cart10_front_temp														:= F_Temperature(_10_TT_01, cart10_front_temp_offset);
cart10_front_temp_error 												:= _10_TT_01_error OR iCount[18] < 30;
cart10_back_temp														:= F_Temperature(_10_TT_03, cart10_back_temp_offset);
cart10_back_temp_error 													:= _10_TT_03_Error OR iCount[19] < 30;
cart10_temp_front_calc(Error:= cart10_front_temp_error, Temp:= cart10_front_temp, Low:= sorbent_low_temp, High:= sorbent_high_temp, Total:= rTempTotal, Counter:= iTempCount);
cart10_temp_back_calc(Error:= cart10_back_temp_error, Temp:= cart10_back_temp, Low:= sorbent_low_temp, High:= sorbent_high_temp, Total:= rTempTotal, Counter:= iTempCount);

cart11_front_temp														:= F_Temperature(_11_TT_01, cart11_front_temp_offset);
cart11_front_temp_error 												:= _11_TT_01_error OR iCount[20] < 30;
cart11_back_temp														:= F_Temperature(_11_TT_03, cart11_back_temp_offset);
cart11_back_temp_error 													:= _11_TT_03_Error OR iCount[21] < 30;
cart11_temp_front_calc(Error:= cart11_front_temp_error, Temp:= cart11_front_temp, Low:= sorbent_low_temp, High:= sorbent_high_temp, Total:= rTempTotal, Counter:= iTempCount);
cart11_temp_back_calc(Error:= cart11_back_temp_error, Temp:= cart11_back_temp, Low:= sorbent_low_temp, High:= sorbent_high_temp, Total:= rTempTotal, Counter:= iTempCount);

cart12_front_temp														:= F_Temperature(_12_TT_01, cart12_front_temp_offset);
cart12_front_temp_error 												:= _12_TT_01_error OR iCount[22] < 30;
cart12_back_temp														:= F_Temperature(_12_TT_03, cart12_back_temp_offset);
cart12_back_temp_error 													:= _12_TT_03_Error OR iCount[23] < 30;
cart12_temp_front_calc(Error:= cart12_front_temp_error, Temp:= cart12_front_temp, Low:= sorbent_low_temp, High:= sorbent_high_temp, Total:= rTempTotal, Counter:= iTempCount);
cart12_temp_back_calc(Error:= cart12_back_temp_error, Temp:= cart12_back_temp, Low:= sorbent_low_temp, High:= sorbent_high_temp, Total:= rTempTotal, Counter:= iTempCount);

sorbent_average_temp													:= SEL(iTempCount > 0, 0, rTempTotal / iTempCount);

FOR i:= 0 TO 23 DO
	iCount[i]															:= iCount[i] + 1;
	IF iCount[i] > 30 THEN
		iCount[i]														:= 30;
	END_IF
END_FOR

iHighTempCount															:= 0;
rMin																	:= P_U01.SP_minimum_reasonable_sorbent_TC_reading;
rMax																	:= P_U01.SP_maximum_reasonable_sorbent_TC_reading;
IF iInletAirSetpoint = 0 THEN
	rTempSP																:= P_M01.SP_vacuum_cooling_target_temperature;
ELSIF iInletAirSetpoint = 1 THEN
	rTempSP																:= P_M01.SP_maximum_inlet_air_temperature_during_adsorption;
ELSE
	rTempSP																:= P_M01.SP_maximum_sorbent_temperature_during_desorption;
END_IF

IF _01_TT_01_Error OR cart01_front_temp < rMin OR cart01_front_temp > rMax THEN
	iCount[0]															:= 0;
ELSIF cart01_front_temp > rTempSP THEN
	iHighTempCount														:= iHighTempCount + 1;
END_IF 
IF _01_TT_03_Error OR cart01_back_temp < rMin OR cart01_back_temp > rMax THEN
	iCount[1]															:= 0;
ELSIF cart01_back_temp > rTempSP THEN
	iHighTempCount														:= iHighTempCount + 1;
END_IF

IF _02_TT_01_Error OR cart02_front_temp < rMin OR cart02_front_temp > rMax THEN
	iCount[2]															:= 0;
ELSIF cart02_front_temp > rTempSP THEN
	iHighTempCount														:= iHighTempCount + 1;
END_IF 
IF _02_TT_03_Error OR cart02_back_temp < rMin OR cart02_back_temp > rMax THEN
	iCount[3]															:= 0;
ELSIF cart02_back_temp > rTempSP THEN
	iHighTempCount														:= iHighTempCount + 1;
END_IF

IF _03_TT_01_Error OR cart03_front_temp < rMin OR cart03_front_temp > rMax THEN
	iCount[4]															:= 0;
ELSIF cart03_front_temp > rTempSP THEN
	iHighTempCount														:= iHighTempCount + 1;
END_IF 
IF _03_TT_03_Error OR cart03_back_temp < rMin OR cart03_back_temp > rMax THEN
	iCount[5]															:= 0;
ELSIF cart03_back_temp > rTempSP THEN
	iHighTempCount														:= iHighTempCount + 1;
END_IF

IF _04_TT_01_Error OR cart04_front_temp < rMin OR cart04_front_temp > rMax THEN
	iCount[6]															:= 0;
ELSIF cart04_front_temp > rTempSP THEN
	iHighTempCount														:= iHighTempCount + 1;
END_IF 
IF _04_TT_03_Error OR cart04_back_temp < rMin OR cart04_back_temp > rMax THEN
	iCount[7]															:= 0;
ELSIF cart04_back_temp > rTempSP THEN
	iHighTempCount														:= iHighTempCount + 1;
END_IF

IF _05_TT_01_Error OR cart05_front_temp < rMin OR cart05_front_temp > rMax THEN
	iCount[8]															:= 0;
ELSIF cart05_front_temp > rTempSP THEN
	iHighTempCount														:= iHighTempCount + 1;
END_IF 
IF _05_TT_03_Error OR cart05_back_temp < rMin OR cart05_back_temp > rMax THEN
	iCount[9]															:= 0;
ELSIF cart05_back_temp > rTempSP THEN
	iHighTempCount														:= iHighTempCount + 1;
END_IF

IF _06_TT_01_Error OR cart06_front_temp < rMin OR cart06_front_temp > rMax THEN
	iCount[10]															:= 0;
ELSIF cart06_front_temp > rTempSP THEN
	iHighTempCount														:= iHighTempCount + 1;
END_IF 
IF _06_TT_03_Error OR cart06_back_temp < rMin OR cart06_back_temp > rMax THEN
	iCount[11]															:= 0;
ELSIF cart06_back_temp > rTempSP THEN
	iHighTempCount														:= iHighTempCount + 1;
END_IF

IF _07_TT_01_Error OR cart07_front_temp < rMin OR cart07_front_temp > rMax THEN
	iCount[12]															:= 0;
ELSIF cart07_front_temp > rTempSP THEN
	iHighTempCount														:= iHighTempCount + 1;
END_IF 
IF _07_TT_03_Error OR cart07_back_temp < rMin OR cart07_back_temp > rMax THEN
	iCount[13]															:= 0;
ELSIF cart07_back_temp > rTempSP THEN
	iHighTempCount														:= iHighTempCount + 1;
END_IF

IF _08_TT_01_Error OR cart08_front_temp < rMin OR cart08_front_temp > rMax THEN
	iCount[14]															:= 0;
ELSIF cart08_front_temp > rTempSP THEN
	iHighTempCount														:= iHighTempCount + 1;
END_IF 
IF _08_TT_03_Error OR cart08_back_temp < rMin OR cart08_back_temp > rMax THEN
	iCount[15]															:= 0;
ELSIF cart08_back_temp > rTempSP THEN
	iHighTempCount														:= iHighTempCount + 1;
END_IF

IF _09_TT_01_Error OR cart09_front_temp < rMin OR cart09_front_temp > rMax THEN
	iCount[16]															:= 0;
ELSIF cart09_front_temp > rTempSP THEN
	iHighTempCount														:= iHighTempCount + 1;
END_IF 
IF _09_TT_03_Error OR cart09_back_temp < rMin OR cart09_back_temp > rMax THEN
	iCount[17]															:= 0;
ELSIF cart09_back_temp > rTempSP THEN
	iHighTempCount														:= iHighTempCount + 1;
END_IF

IF _10_TT_01_Error OR cart10_front_temp < rMin OR cart10_front_temp > rMax THEN
	iCount[18]															:= 0;
ELSIF cart10_front_temp > rTempSP THEN
	iHighTempCount														:= iHighTempCount + 1;
END_IF 
IF _10_TT_03_Error OR cart10_back_temp < rMin OR cart10_back_temp > rMax THEN
	iCount[19]															:= 0;
ELSIF cart10_back_temp > rTempSP THEN
	iHighTempCount														:= iHighTempCount + 1;
END_IF

IF _11_TT_01_Error OR cart11_front_temp < rMin OR cart11_front_temp > rMax THEN
	iCount[20]															:= 0;
ELSIF cart11_front_temp > rTempSP THEN
	iHighTempCount														:= iHighTempCount + 1;
END_IF 
IF _11_TT_03_Error OR cart11_back_temp < rMin OR cart11_back_temp > rMax THEN
	iCount[21]															:= 0;
ELSIF cart11_back_temp > rTempSP THEN
	iHighTempCount														:= iHighTempCount + 1;
END_IF

IF _12_TT_01_Error OR cart12_front_temp < rMin OR cart12_front_temp > rMax THEN
	iCount[22]															:= 0;
ELSIF cart12_front_temp > rTempSP THEN
	iHighTempCount														:= iHighTempCount + 1;
END_IF 
IF _12_TT_03_Error OR cart12_back_temp < rMin OR cart12_back_temp > rMax THEN
	iCount[23]															:= 0;
ELSIF cart12_back_temp > rTempSP THEN
	iHighTempCount														:= iHighTempCount + 1;
END_IF

IF iInletAirSetpoint = 0 THEN
	vacuum_cooling_high_temp_count										:= iHighTempCount;
ELSIF iInletAirSetpoint = 1 THEN
	adsorption_high_temp_count											:= iHighTempCount;
ELSE
	desorption_high_temp_count											:= iHighTempCount;
END_IF
iInletAirSetpoint														:= SEL(iInletAirSetpoint = 2, iInletAirSetpoint + 1, 0);;
END_ACTION

END_FUNCTION_BLOCK

// ---- POUs/Function_Blocks/FB_VFD.TcPOU
FUNCTION_BLOCK FB_VFD
VAR_INPUT
	Enable_Vfd															: BOOL;
	Fault_Reset															: BOOL;
	Rpm																	: REAL;
	Minimum_Speed														: REAL		:= 0;
	Maximum_Speed														: REAL		:= 1800;
	StatusWord															: WORD;
END_VAR
VAR_OUTPUT
	ControlWord															: WORD;
	TargetRpm															: WORD;
	Ready																: BOOL;
	Error																: BOOL;
END_VAR
VAR
	rtrigClear															: R_TRIG;
	rtrigReady															: R_TRIG;
	rtrigRun															: R_TRIG;
	tonReady															: TON;
	tonRun																: TON;
	rRpm																: REAL;
	bEnabled															: BOOL;
	
	VFD_OFF																: WORD										:= 0;
	VFD_CLEAR															: WORD										:= 6;
	VFD_READY															: WORD										:= 7;
	VFD_RUN																: WORD										:= 15;
	VFD_FAULTED															: WORD										:= 8;
	VFD_RESET															: WORD										:= 128;
END_VAR

//// FB_VFD
//// Rev 1.0 - April 11, 2024

// Need to add parse status word

rRpm := Rpm;

bEnabled																:= Enable_Vfd;
IF rRpm = 0 THEN
	bEnabled															:= FALSE;											// Turn output off if rpm is 0
ELSIF rRpm > Maximum_Speed THEN
	rRpm																:= Maximum_Speed;
ELSIF rRpm < Minimum_Speed THEN
	rRpm																:= Minimum_Speed;
END_IF

rtrigClear(CLK:= bEnabled);
IF rtrigClear.Q THEN
	ControlWord															:= VFD_CLEAR;
END_IF

rtrigReady(CLK:= tonReady.Q);
IF rtrigReady.Q THEN
	ControlWord															:= VFD_READY;
END_IF
tonReady(IN:= ControlWord = VFD_CLEAR, PT:= T#100MS);

rtrigRun(CLK:= tonRun.Q);
IF rtrigRun.Q THEN
	ControlWord															:= VFD_RUN;
END_IF
tonRun(IN:= ControlWord = VFD_READY, PT:= T#100MS);

IF NOT bEnabled AND NOT Fault_Reset THEN
	ControlWord															:= VFD_OFF;
	rtrigReady(CLK:= FALSE);
END_IF

IF Error AND Fault_Reset THEN
	ControlWord															:= VFD_RESET;
END_IF

Ready																	:= ControlWord = VFD_READY OR ControlWord = VFD_RUN OR Enable_Vfd;
TargetRpm																:= SEL(Ready, 0, REAL_TO_WORD(rRpm));

Error																	:= (StatusWord AND VFD_FAULTED) > 0;

END_FUNCTION_BLOCK

// ---- POUs/Function_Blocks/FB_Door_Closed.TcPOU
FUNCTION_BLOCK FB_Door_Closed
VAR_INPUT
	valve																: BOOL;
	limit_switch														: BOOL;
END_VAR
VAR_OUTPUT
	door_closed															: BOOL;
END_VAR
VAR
	ton1																: TON;
	rtrig1																: R_TRIG;
END_VAR

// FB_Door_Closed
// Rev 1.0 - November 2, 2024

ton1(IN:= valve AND limit_switch, PT:= _DOOR_LATCH_CLOSE_TIME);
rtrig1(CLK:= ton1.Q);
IF rtrig1.Q THEN
	door_closed															:= TRUE;
ELSIF NOT valve THEN
	door_closed															:= FALSE;
END_IF

END_FUNCTION_BLOCK

// ---- POUs/Function_Blocks/FB_Temperature.TcPOU
FUNCTION_BLOCK FB_Temperature
VAR_INPUT
	Error																: BOOL;
	Temp																: REAL;
	Low																	: REFERENCE TO REAL;
	High																: REFERENCE TO REAL;
	Total																: REFERENCE TO REAL;
	Counter																: REFERENCE TO INT;
END_VAR
VAR
END_VAR

// Theseus - FB_Temperature
// Rev 1.0 - April 25, 2024

IF NOT Error THEN
	Low																	:= F_LowestReal(Temp, Low);
	High																:= F_HighestReal(Temp, High, 0, 0);
	Total																:= Total + Temp;
	Counter																:= Counter + 1;
END_IF

END_FUNCTION_BLOCK

// ---- POUs/Functions/F_HighestReal.TcPOU
FUNCTION F_HighestReal : REAL
VAR_INPUT
	Value1																: REAL;
	Value2																: REAL;
	Value3																: REAL;
	Value4																: REAL;
END_VAR
VAR
	rValue																: REAL;
END_VAR

// F_HighestReal
// Rev 1.0 - April 25, 2024

rValue																		:= SEL(Value1 > Value2, Value2, Value1);
rValue																		:= SEL(rValue > Value3, Value3, rValue);
F_HighestReal																:= SEL(rValue > Value4, Value4, rValue);

END_FUNCTION

// ---- POUs/MAIN.TcPOU
PROGRAM MAIN
VAR
	bHalfSecondPulse													: BOOL;
	tonHalfSecPulse														: TON;
END_VAR

// Theseus - Main
// Rev 1.0 - September 31, 2024

P_M01.plc_version														:= '24_12_03_00';

/// TIMER PULSE
IF tonHalfSecPulse.Q THEN
	bHalfSecondPulse													:= NOT bHalfSecondPulse;
	tonHalfSecPulse(IN:= FALSE);
END_IF
tonHalfSecPulse(IN:= TRUE, PT:= T#500MS);

P_U01();
P_M01();
P_Alarms();

END_PROGRAM

// ---- POUs/P_M01.TcPOU
PROGRAM P_M01
VAR_INPUT
	rs1																	: FB_Reactor_Set();
	stop_rs																: BOOL;
	clear_rs															: BOOL;
	
	{attribute 'OPC.UA.DA' := '1'}  				                
	{attribute 'OPC.UA.DA.Access' := '1'}  				                
	plc_version															: STRING;
	{attribute 'OPC.UA.DA' := '1'}  				                
	{attribute 'OPC.UA.DA.Access' := '1'}  				                
	tb_Alarm_Active														: BOOL;			// An alarm is active
	{attribute 'OPC.UA.DA' := '1'}  				                
	{attribute 'OPC.UA.DA.Access' := '1'}  				                
	ts_Alarm															: STRING;		// Active alarm string
	{attribute 'OPC.UA.DA' := '1'}  				                
	{attribute 'OPC.UA.DA.Access' := '1'}  				                
	ts_User_Message														: STRING;		// Message corresponding to active alarm
	{attribute 'OPC.UA.DA' := '1'}  				                
	{attribute 'OPC.UA.DA.Access' := '1'}  				                
	ti_Alarm_Severity													: INT;			// Alarm level (not implemented)	
	{attribute 'OPC.UA.DA' := '1'}  
	processAlarms														: ARRAY[0.._ALARM_COUNT] OF STRING;
	{attribute 'OPC.UA.DA' := '1'}  
	processAlarmsMessage												: ARRAY[0.._ALARM_COUNT] OF STRING;
	{attribute 'OPC.UA.DA' := '1'}  				                
	tb_Acknowledge_Alarm												: BOOL;			// Clears current alarm
	{attribute 'OPC.UA.DA' := '1'}  				                
	tb_Clear_Alarm_All													: BOOL;			// Clears current alarm
END_VAR
VAR
	sCycleModeRS01														: STRING	:= '';
	iRS01CyclesToRun													: INT;
	iLength																: INT;
	iRS01Count															: INT;
	rtrigStart															: R_TRIG;
	
	bRSProcess															: BOOL;
	bRSManual															: BOOL;
	bRS01																: BOOL;
	bRS01Selected														: BOOL;
	bStarted															: BOOL;
	bReactorSetSelected													: BOOL;
	
	rtrigRS01StartNextRS												: R_TRIG;
	rtrigRS01Restart													: R_TRIG;
	rtrigRS01Done														: R_TRIG;
	rtrigRS01Offline													: R_TRIG;
	
	rtrigCPDrainLSHOn													: R_TRIG;
	tonCPDrainErrorOn													: TON;
	tonCPDrainErrorOff													: TON;
	bCPDrainError														: BOOL;
	
	rMinPressureSP														: REAL; 
	rMaxPressureSP														: REAL;
	
	{attribute 'OPC.UA.DA' := '1'}  				                
	ts_Cycle_Mode														: STRING;		// Starts process based on each character in integer format
	{attribute 'OPC.UA.DA' := '1'}  				                
	tb_HMI_Active														: BOOL;			// An HMI program is running and communicating
	{attribute 'OPC.UA.DA' := '1'}  				                
	tb_Cancel_Cycle														: BOOL;			// Complete current cycle then stop
	{attribute 'OPC.UA.DA' := '1'}  				                
	tb_Stop_Process														: BOOL;			// Stop current process immediately
	{attribute 'OPC.UA.DA' := '1'}  				                
	tb_Reset_Process													: BOOL;
	
					
	{attribute 'OPC.UA.DA' := '1'}  				                
	{attribute 'OPC.UA.DA.Access' := '1'}  				                
	tb_Auto_Mode_On														: BOOL;			// Machine is currently in auto mode

END_VAR

VAR PERSISTENT

	/// SET POINTS

	{attribute 'OPC.UA.DA' := '1'}
	SP_evacuation_ideal_pressure										: REAL;
	{attribute 'OPC.UA.DA' := '1'}
	SP_evacuation_duration												: REAL;
	{attribute 'OPC.UA.DA' := '1'}
	SP_vacuum_settle_time												: REAL;
	{attribute 'OPC.UA.DA' := '1'}
	SP_vacuum_leak_test_duration										: REAL;
	{attribute 'OPC.UA.DA' := '1'}
	SP_unacceptable_vacuum_pressure_change								: REAL;
	{attribute 'OPC.UA.DA' := '1'}
	SP_pos_pres_ideal_pressure											: REAL;		
	{attribute 'OPC.UA.DA' := '1'}
	SP_pos_pres_settle_time												: REAL;		
	{attribute 'OPC.UA.DA' := '1'}
	SP_pos_pres_leak_test_duration										: REAL;		
	{attribute 'OPC.UA.DA' := '1'}
	SP_unacceptable_pos_pres_change										: REAL;		

	
	{attribute 'OPC.UA.DA' := '1'}
	SP_adsorption_sorbent_hightemp_startco2analyzer						: REAL;		
	{attribute 'OPC.UA.DA' := '1'}
	SP_adsorption_outletco2_highlimit									: REAL;		
	{attribute 'OPC.UA.DA' := '1'}
	SP_repres_preslimit_clampsretract									: REAL;		
	{attribute 'OPC.UA.DA' := '1'}
	SP_clampsretract_timedelay											: REAL;		
	{attribute 'OPC.UA.DA' := '1'}
	SP_repres_pres_highlimit											: REAL;		
	{attribute 'OPC.UA.DA' := '1'}
	SP_doorsopenclose_timedelay											: REAL;		
	{attribute 'OPC.UA.DA' := '1'}
	SP_adsorption_duration												: REAL;
	{attribute 'OPC.UA.DA' := '1'}
	SP_adsorption_valve_max_retries										: INT;		
	{attribute 'OPC.UA.DA' := '1'}
	SP_adsorption_valve_rotational_velocity								: REAL;		
	{attribute 'OPC.UA.DA' := '1'}
	SP_ambient_pressure													: REAL;
	{attribute 'OPC.UA.DA' := '1'}
	SP_cycle_start_offset_duration										: REAL;
	{attribute 'OPC.UA.DA' := '1'}
	SP_dead_time_in_cycle_duration										: REAL;
	{attribute 'OPC.UA.DA' := '1'}
	SP_desired_cycle_count												: INT;
	{attribute 'OPC.UA.DA' := '1'}
	SP_evacuation_unacceptable_pressure									: REAL;
	{attribute 'OPC.UA.DA' := '1'}
	SP_include_reactor_set_1_in_process									: BOOL;					
	{attribute 'OPC.UA.DA' := '1'}
	SP_include_reactor_set_2_in_process									: BOOL;
	{attribute 'OPC.UA.DA' := '1'}
	SP_include_reactor_set_3_in_process									: BOOL;	
	{attribute 'OPC.UA.DA' := '1'}
	SP_initial_maximum_steam_valve_percent_open							: REAL;
	{attribute 'OPC.UA.DA' := '1'}
	SP_initial_steam_purge_reactor_pressure								: REAL;
	{attribute 'OPC.UA.DA' := '1'}
	SP_leak_test_duration												: REAL;
	{attribute 'OPC.UA.DA' := '1'}
	SP_maximum_desorption_starting_pressure								: REAL;							
	{attribute 'OPC.UA.DA' := '1'}
	SP_maximum_inlet_air_temperature_during_adsorption					: REAL;						
	{attribute 'OPC.UA.DA' := '1'}
	SP_maximum_reactor_leakage_pressure									: REAL;												// PS 11/27/24
	{attribute 'OPC.UA.DA' := '1'}
	SP_maximum_reactor_pressure_to_introduce_steam						: REAL;												// PS 08_12_24
	{attribute 'OPC.UA.DA' := '1'}
	SP_maximum_safe_ambient_temperature									: REAL;												// PS 08_12_24
	{attribute 'OPC.UA.DA' := '1'}
	SP_maximum_safe_co2_adsorption_sensor_temperature					: REAL;												// PS 08_16_24
	{attribute 'OPC.UA.DA' := '1'}
	SP_maximum_safe_reactor_steam_pressure								: REAL;
	{attribute 'OPC.UA.DA' := '1'}
	SP_maximum_safe_sorbent_temperature									: REAL;												// PS 08_15_24
	{attribute 'OPC.UA.DA' := '1'}
	SP_maximum_sorbent_temperature_during_desorption					: REAL;			
	{attribute 'OPC.UA.DA' := '1'}
	SP_maximum_sorbent_temperature_to_use_dead_air_line					: REAL;												// PS 08_12_24			
	{attribute 'OPC.UA.DA' := '1'}
	SP_maximum_target_sorbent_temperature_during_purge					: REAL;												// PS 04_25_24			
	{attribute 'OPC.UA.DA' := '1'}
	SP_maximum_target_sorbent_temperature_to_repressurize				: REAL;												// PS 08_15_24		
	{attribute 'OPC.UA.DA' := '1'}
	SP_maximum_target_steam_pressure									: REAL;			
	{attribute 'OPC.UA.DA' := '1'}
	SP_minimum_desired_inlet_co2_concentration_during_adsorption		: REAL;						
	{attribute 'OPC.UA.DA' := '1'}
	SP_minimum_inlet_air_temperature_during_adsorption					: REAL;						
	{attribute 'OPC.UA.DA' := '1'}
	SP_module_steam_line_high_pressure									: REAL;
	{attribute 'OPC.UA.DA' := '1'}
	SP_module_steam_line_high_temperature								: REAL;
	{attribute 'OPC.UA.DA' := '1'}
	SP_module_steam_line_low_pressure									: REAL;
	{attribute 'OPC.UA.DA' := '1'}
	SP_module_steam_line_low_temperature								: REAL;
	{attribute 'OPC.UA.DA' := '1'}
	SP_percent_from_steam_purge_target_pressure							: REAL;
	{attribute 'OPC.UA.DA' := '1'}
	SP_percent_of_ambient_pressure										: REAL;
	{attribute 'OPC.UA.DA' := '1'}
	SP_reactor_set_1_vfd_percent										: INT;
	{attribute 'OPC.UA.DA' := '1'}
	SP_reactor_set_2_vfd_percent										: INT;
	{attribute 'OPC.UA.DA' := '1'}
	SP_reactor_set_3_vfd_percent										: INT;
	{attribute 'OPC.UA.DA' := '1'}
	SP_repressurization_duration										: REAL;
	{attribute 'OPC.UA.DA' := '1'}
	SP_start_steam_purge_reactor_pressure								: REAL;
	{attribute 'OPC.UA.DA' := '1'}
	SP_steam_pressure_control_valve_initial_opening_duration			: REAL;					
	{attribute 'OPC.UA.DA' := '1'}
	SP_steam_pressurization_and_purge_duration							: REAL;						
	{attribute 'OPC.UA.DA' := '1'}
	SP_steam_purge_pressure												: REAL;
	{attribute 'OPC.UA.DA' := '1'}
	SP_steam_purge_pressure_decrease									: REAL;												// PS 04_25_24
	{attribute 'OPC.UA.DA' := '1'}
	SP_target_desorption_starting_pressure								: REAL;
	{attribute 'OPC.UA.DA' := '1'}
	SP_target_duration_from_adsorption_start_until_sorbent_cool			: REAL;							
	{attribute 'OPC.UA.DA' := '1'}
	SP_target_pressure_change											: REAL;
	{attribute 'OPC.UA.DA' := '1'}
	SP_unacceptable_duration_from_adsorption_start_until_sorbent_cool	: REAL;					
	{attribute 'OPC.UA.DA' := '1'}
	SP_undesirable_duration_from_adsorption_start_until_sorbent_cool	: REAL;
	{attribute 'OPC.UA.DA' := '1'}
	SP_vacuum_assisted_purge											: BOOL;
	{attribute 'OPC.UA.DA' := '1'}
	SP_vacuum_cooling_duration											: REAL;
	{attribute 'OPC.UA.DA' := '1'}
	SP_vacuum_cooling_target_pressure									: REAL;
	{attribute 'OPC.UA.DA' := '1'}
	SP_vacuum_cooling_target_temperature								: REAL;
	{attribute 'OPC.UA.DA' := '1'}
	SP_vacuum_cooling_unacceptable_pressure								: REAL;
	{attribute 'OPC.UA.DA' := '1'}
	SP_vacuum_cooling_unacceptable_temperature							: REAL;
	{attribute 'OPC.UA.DA' := '1'}
	SP_extend_wallace_clamp_duration									: REAL;
			
END_VAR

// Theseus - P_M01
// Rev 1.0 - November 27, 2024

A_Drain_Condensate_Product_Cooling_Lines();

rs1(	stop_rs_automode												:= stop_rs,
        clear_reactor_set_pause											:= clear_rs);
		
rMinPressureSP															:= SP_ambient_pressure - (SP_percent_of_ambient_pressure / 100 * SP_ambient_pressure); 
rMaxPressureSP															:= SP_ambient_pressure + (SP_percent_of_ambient_pressure / 100 * SP_ambient_pressure);

A_AutoMode();

ACTION A_AutoMode:
// Theseus - P_M01.A_AutoMode
// Rev 1.0 - October 4, 2024

IF tb_Stop_Process OR rs1.utility_error THEN 																	// Stop all processes from HMI or if utility error occurs
	P_U01.shutdown_process												:= TRUE;
//	rs1.stop_rs_automode												:= TRUE;
	stop_rs																:= TRUE;
	bRSProcess															:= FALSE;
	tb_Stop_Process														:= FALSE;
END_IF

IF tb_Cancel_Cycle OR rs1.cancel_all_reactor_sets THEN
	iRS01CyclesToRun													:= SEL(rs1.tb_Process_Running, iRS01Count, iRS01Count + 1);
	bRS01																:= SEL(iRS01Count >= iRS01CyclesToRun, bRS01, FALSE);
	tb_Cancel_Cycle														:= FALSE;
END_IF

A_AutoMode_RS01();

bReactorSetSelected														:= SP_include_reactor_set_1_in_process;
IF ts_Cycle_Mode <> '' AND (P_U01.sUtilityError <> '' OR SP_desired_cycle_count = 0 OR NOT bReactorSetSelected) THEN		// Don't allow cycle if moodule or utility error occured, cycle count is zero or no reactor sets are selected
	IF P_U01.sUtilityError  <> '' THEN
		P_Alarms.M_Add_Alarm(_U01, P_U01.sUtilityError, gsProcessCannotRun);
	ELSIF SP_desired_cycle_count = 0 THEN
		P_Alarms.M_Add_Alarm(_U01, gsDesiredCycleCountError, gsProcessCannotRun);
	ELSE
		P_Alarms.M_Add_Alarm(_U01, gsNoReactorSetsSelected, gsProcessCannotRun);
	END_IF
	ts_Cycle_Mode														:= '';
END_IF

iLength																	:= LEN(ts_Cycle_Mode);							// Start process in this order '6745' (Evac, Desorp, Repres, Adsorp)
rtrigStart(CLK:= iLength > 0);
IF rtrigStart.Q THEN
	gsCycleMode															:= ts_Cycle_Mode;
	ts_Cycle_Mode														:= '';
	iRS01CyclesToRun													:= SP_desired_cycle_count;
	bRS01																:= SP_include_reactor_set_1_in_process;			// Get active reactors
	IF iLength = 1 THEN																										// Single process selected
		tb_Auto_Mode_On													:= FALSE;
		bRSManual														:= STRING_TO_INT(gsCycleMode) >= eDoorCycle AND STRING_TO_INT(gsCycleMode) <= eDesorption;
	ELSE
		bRS01Selected													:= bRS01;
		rs1.ti_Cycle_Count												:= 0;												// Completed cycles
		iRS01Count														:= 0;												// Attempted cycles
		tb_Auto_Mode_On													:= TRUE;
		bRSProcess														:= TRUE;
	END_IF
END_IF

IF bRSManual THEN
	sCycleModeRS01														:= SEL(bRS01, sCycleModeRS01, gsCycleMode);
	bRSManual															:= FALSE;
ELSIF bRSProcess THEN
	IF NOT bStarted THEN
		sCycleModeRS01													:= gsCycleMode;
		bStarted														:= TRUE;
	END_IF
	IF NOT bRS01 THEN																										// Stop process if reactor is not selected
//		rs1.stop_rs_automode											:= TRUE;
		stop_rs															:= TRUE;
		bRSProcess														:= FALSE;
	END_IF
	
	rtrigRS01Done(CLK:= rs1.Done);
	IF rtrigRS01Done.Q THEN
		sCycleModeRS01													:= '';												// Turn off cycle
		bStarted														:= FALSE;
		iRS01Count														:= iRS01Count + 1;									// This counter increments regardless of reactor status if long as reactor was selected
		IF iRS01Count >= iRS01CyclesToRun THEN
			bRS01														:= FALSE;
			gsCycleMode													:= '';
		END_IF
		IF rs1.tb_Process_Complete THEN 																				// Increment counter once a valid cycle has run
			rs1.ti_Cycle_Count											:= rs1.ti_Cycle_Count + 1;
			rs1.ti_Total_Cycle_Count									:= 1;			///@@@
		END_IF
	END_IF
	
ELSE
//	P_U01.write_persistent_data											:= TRUE;
	sCycleModeRS01														:= '';
	bRS01																:= FALSE;
	bStarted															:= FALSE;
	tb_Auto_Mode_On														:= FALSE;
	
END_IF

rs1.cycle_mode 															:= sCycleModeRS01;

IF NOT rs1.Process_Running THEN 
	rs1.cycle_stage														:= gsCycleStage;
//	gsCycleMode															:= '';
END_IF

// rs1.cycle_stage															:= SEL(bRS01 AND gsCycleStage <> '', gsM01RS01CycleStage, gsCycleStage);
END_ACTION

ACTION A_AutoMode_RS01:
// Theseus - P_M01.A_AutoMode_RS01
// Rev 1.0 - October 4, 2024

rtrigRS01Restart(CLK:= SP_include_reactor_set_1_in_process);
IF rtrigRS01Restart.Q THEN
	IF tb_Auto_Mode_On AND NOT bRS01Selected THEN 
		SP_include_reactor_set_1_in_process								:= FALSE;
	ELSE
		bRS01															:= TRUE;
		rs1.clear_rs_pause												:= TRUE;
	END_IF
END_IF

//IF rs1.stop_rs_automode THEN
IF stop_rs THEN
	SP_include_reactor_set_1_in_process									:= FALSE;
	bRS01Selected														:= FALSE;
END_IF

rtrigRS01Offline(CLK:= NOT SP_include_reactor_set_1_in_process);
IF rtrigRS01Offline.Q THEN
	bRS01																:= FALSE;
END_IF

IF rs1.cancel_reactor_set THEN
	iRS01CyclesToRun													:= SEL(rs1.tb_Process_Running, iRS01Count, iRS01Count + 1);
END_IF
END_ACTION

ACTION A_Drain_Condensate_Product_Cooling_Lines:
// Theseus - P_M01.A_Drain_Condensate_Product_Cooling_Lines
// Rev 1.0 - June 10, 2024

(*IF gbDrainageOn THEN
	IF (P_U01.purge_product_line_pres < P_U01.SP_drainage_function_cutoff_pressure) OR
		(m01_rs1.purge_valve_closed AND m01_rs1.condensate_valve_closed) THEN
		m.condensate_from_cooling_and_purge_lines_pump					:= FALSE;
	ELSE
		IF m.condensate_from_cooling_and_purge_linesh THEN
			m.condensate_from_cooling_and_purge_lines_pump				:= TRUE;
		END_IF
		IF NOT m.condensate_from_cooling_and_purge_linesl THEN
			m.condensate_from_cooling_and_purge_lines_pump				:= FALSE;
		END_IF
	END_IF
	
	rtrigCPDrainLSHOn(CLK:= tonCPDrainErrorOn.Q);
	IF rtrigCPDrainLSHOn.Q THEN
		P_Alarms.M_Add_Alarm(_M01, gsCondensateProductDrainError, gsProcessStopsAtEOC);
		m.condensate_from_cooling_and_purge_lines_pump					:= FALSE;
		bCPDrainError													:= TRUE;
		m01.tb_Cancel_Cycle												:= TRUE;											// Complete current cycles
	END_IF
	tonCPDrainErrorOn(IN:= m.condensate_from_cooling_and_purge_linesh AND NOT bCPDrainError, PT:= _DRAIN_TIME);
	
	IF tonCPDrainErrorOff.Q THEN
		bCPDrainError													:= FALSE;
	END_IF
	tonCPDrainErrorOff(IN:= NOT m.condensate_from_cooling_and_purge_linesh AND bCPDrainError, PT:= _DRAIN_TIME);
END_IF
*)
END_ACTION

END_PROGRAM

// ---- POUs/FB_Reactor_Set.TcPOU
FUNCTION_BLOCK FB_Reactor_Set
VAR_IN_OUT
	//stop_reactor_set													: BOOL;
	stop_rs_automode													: BOOL;
	clear_reactor_set_pause												: BOOL;
END_VAR
VAR_INPUT
	r1																	: FB_Reactor;
	
	rs_name																: STRING;
	cycle_mode															: STRING;
//	stop_rs_automode													: BOOL;
	clear_rs_pause														: BOOL;
	open_doors															: BOOL;
	close_doors															: BOOL;
	close_valves														: BOOL;
	retract_clamps														: BOOL;
	extend_clamps														: BOOL;
	
	{attribute 'OPC.UA.DA' := '1'}  				                
	fan_setpoint														: REAL;
	{attribute 'OPC.UA.DA' := '1'}  				                
	{attribute 'OPC.UA.DA.Access' := '1'}  				                
	ti_Cycle_Count														: INT; 
	{attribute 'OPC.UA.DA' := '1'}  				                
	{attribute 'OPC.UA.DA.Access' := '1'}  				                
	ti_Total_Cycle_Count												: DINT; 
	{attribute 'OPC.UA.DA' := '1'}  				                
	{attribute 'OPC.UA.DA.Access' := '1'}  				                
	cycle_stage															: STRING;
    /// <summary>RS_XV08</summary>
	{attribute 'OPC.UA.DA' := '1'}  				                
	steam_bypass_valve													: BOOL;
	/// <summary>XV02</summary>
	{attribute 'OPC.UA.DA' := '1'}  	//mm 11/7 to command valve
	repres_valves														: BOOL;
END_VAR
VAR_OUTPUT
	
	inlet_doors_open													: BOOL;
	inlet_doors_closed													: BOOL;
	outlet_doors_open													: BOOL;
	outlet_doors_closed													: BOOL;

	inlet_clamps_extended												: BOOL;
	inlet_clamps_retracted												: BOOL;
	outlet_clamps_extended												: BOOL;
	outlet_clamps_retracted												: BOOL;
	
	rs_valves_clear														: BOOL;
	adsorption_high_temp_count											: INT;
	desorption_high_temp_count											: INT;
	vacuum_cooling_high_temp_count										: INT;
	sorbent_high_temp													: REAL;
	sorbent_average_temp												: REAL;
	
    /// <summary>Reactor XV02</summary>
	repres_valves_clear													: BOOL;
    /// <summary>RS_XV04</summary>
	dead_air_valve_clear												: BOOL;
    /// <summary>RS_XV05</summary>
	product_iso_valve_clear												: BOOL;
    /// <summary>RS_XV06</summary>
	condensate_valve_clear												: BOOL;
    /// <summary>RS_XV07</summary>
	steam_iso_valve_clear												: BOOL;
    /// <summary>RS_XV08</summary>
	steam_bypass_valve_clear											: BOOL;
	
	/// <summary>RS_LS01</summary>
	{attribute 'OPC.UA.DA' := '1'}  				                
	{attribute 'OPC.UA.DA.Access' := '1'}  				                
	reactor_drain_vessel_lsl									AT %I*	: BOOL;
    /// <summary>RS_LS02</summary>
	{attribute 'OPC.UA.DA' := '1'}  				                
	{attribute 'OPC.UA.DA.Access' := '1'}  				                
	reactor_drain_vessel_lsh									AT %I*	: BOOL;

    /// <summary>RS_FT02</summary>
	{attribute 'OPC.UA.DA' := '1'}  				                
	{attribute 'OPC.UA.DA.Access' := '1'}  				                
	reactor_condensate_flow												: REAL;

	Remaining_Time														: REAL;
	Current_Step														: INT;
	Machine_State														: INT;
	Status																: INT;
	Process_Running														: BOOL;
	Pause_Reactor_Set													: BOOL;
	Reactor_Set_Stopped													: BOOL;
	DoorCycle_Running													: BOOL;
	PositivePressure_Running											: BOOL;
	Repressurization_Running											: BOOL;
	Adsorption_Running													: BOOL;
	Evacuation_Running													: BOOL;
	Desorption_Running													: BOOL;
	Bypass_Running														: BOOL;
	Utility_Error														: BOOL;
	Cancel_Reactor_Set													: BOOL;
	Cancel_All_Reactor_Sets												: BOOL;
	Process_Complete													: BOOL;
	Done																: BOOL;
	
END_VAR
VAR
	eState																: E_MachineState;
	i																	: INT;
	iStatePointer														: INT;
	iLength																: INT;
	iStateMode															: ARRAY[0..9] OF INT;
	stop_reactor_set													: BOOL;
	
	sUtilityError														: STRING;
	sReactorError														: STRING;
	sCancelError														: STRING;
	sRetryError															: STRING;
	sError																: STRING;
	sMessage															: STRING;
	sLeakageAcceptable													: STRING;
	sLeakageUnacceptable												: STRING;

	rAveragePressure													: REAL;
	iCount																: INT;
	iVacuumStatus														: INT;
	iError																: INT;
	
	rTime																: REAL;
	rTime1																: REAL;
	rTime2																: REAL;
	rTime3																: REAL;
	rSP1																: REAL;
	rSP2																: REAL;
	rSP3																: REAL;
	rR1SavedPressure													: REAL;
	rR1Leakage															: REAL;
	rIncrementalMove													: REAL;
	rPosition															: REAL;
	rAverageReactorPres													: REAL;
	rReactorLeakTestStartingPressure									: REAL;
	
	tTime																: TIME;
	
	iStep																: INT;
	i2Step																: INT;
	i3Step																: INT;
	i4Step																: INT;
	i5Step																: INT;
	i6Step																: INT;
	i7Step																: INT;
	i8Step																: INT;
	iStartStep															: INT;
	iStatus																: INT;
	iErrorProcess														: INT;
	iR1Leakage															: INT;
	iCycleCount															: INT;
	iMaxSorbentTempErrorCount											: INT;

	bMultiProcess														: BOOL;
	bEndProcess															: BOOL;
	bSPAdjust															: BOOL;
	bPaused																: BOOL;
	bClearingCycle														: BOOL;
	bDoorCycleDone								        				: BOOL;
	bPositivePressureDone						        				: BOOL;
	bRepressurizationDone												: BOOL;
	bAdsorptionDone														: BOOL;
	bEvacuationDone														: BOOL;
	bDesorptionDone									        			: BOOL;
	bBypassDone									        				: BOOL;
	bPass1																: BOOL;
	bPass2																: BOOL;
	bPass3																: BOOL;
	bPass4																: BOOL;
	bPass5																: BOOL;
	bPass6																: BOOL;
	bPass7																: BOOL;
	bPass8																: BOOL;
	bPass9																: BOOL;
	bPass10																: BOOL;
	
	
	bCondenserKnockoutOn												: BOOL;
	bStop																: BOOL;
	bTimer1																: BOOL;
	bTimer2																: BOOL;
	bTimer3																: BOOL;
	bRunning															: BOOL;
	bDrainError															: BOOL;
	bPumpOn																: BOOL;
	bPumpTimeOut														: BOOL;									
	bDrainResetToLSL													: BOOL;
	bProcessStarted														: BOOL;
	bDesorptionErrorCheck												: BOOL;
	bSafeShutdownOn														: BOOL;
	bInletClampsRetracted												: BOOL;
	bInletClampsExtended												: BOOL;
	bOutletClampsRetracted												: BOOL;
	bOutletClampsExtended												: BOOL;
	bVacuumHolding														: BOOL;
	bCondition21														: BOOL;
	bCondition22														: BOOL;
	bCondition11														: BOOL;
	bCondition12														: BOOL;
	
	rtrigStart															: R_TRIG;
	rtrigPaused															: R_TRIG;
	rtrigIdle															: R_TRIG;
	rtrigDoorCycle														: R_TRIG;
	rtrigPositivePressure												: R_TRIG;
	rtrigRepressurization												: R_TRIG;
	rtrigAdsorption														: R_TRIG;
	rtrigEvacuation														: R_TRIG;
	rtrigDesorption														: R_TRIG;
	rtrigBypass															: R_TRIG;
	rtrigSingleProcessAuto												: R_TRIG;
	rtrigDrainLSHOn														: R_TRIG;
	
	tonTimer1															: TON;
	tonTimer2															: TON;
	tonTimer3															: TON;
	tonPause															: TON;
	tonDrain															: TON;
	rtrigCondensateValveOff_DrainOff									: R_TRIG;
	tonProcess															: TON;
	
	tRestartTime														: TIME;

	bSteamHeaderValve													: BOOL;
	bCondition1															: BOOL;
	bCondition2															: BOOL;
	bCondition3															: BOOL;
	
	reactor_drain_adsorption_on											: BOOL;
	tmrDrainAdsorp														: TON;
	waterscale_desorp													: REAL;
	water_scale_change_oor												: BOOL;
	fb_adsorp_reactor_wastewater											: FB_ChangeOfValue;
	
	
	{attribute 'OPC.UA.DA' := '1'}  				                
	{attribute 'OPC.UA.DA.Access' := '1'}  				                
	ti_Machine_State													: INT;
	{attribute 'OPC.UA.DA' := '1'}  				                
	{attribute 'OPC.UA.DA.Access' := '1'}  				                
	ti_Current_Step														: INT;
	{attribute 'OPC.UA.DA' := '1'}  				                
	{attribute 'OPC.UA.DA.Access' := '1'}  				                
	tb_Process_Running													: BOOL;
	{attribute 'OPC.UA.DA' := '1'}  				                
	{attribute 'OPC.UA.DA.Access' := '1'}  				                
	tb_Repressurization_Running											: BOOL;
	{attribute 'OPC.UA.DA' := '1'}  				                
	{attribute 'OPC.UA.DA.Access' := '1'}  				                
	tb_Adsorption_Running												: BOOL;
	{attribute 'OPC.UA.DA' := '1'}  				                
	{attribute 'OPC.UA.DA.Access' := '1'}  				                
	tb_Evacuation_Running												: BOOL;
	{attribute 'OPC.UA.DA' := '1'}  				                
	{attribute 'OPC.UA.DA.Access' := '1'}  				                
	tb_Desorption_Running												: BOOL;
	{attribute 'OPC.UA.DA' := '1'}  				                
	{attribute 'OPC.UA.DA.Access' := '1'}  				                
	tb_Bypass_Running													: BOOL;
	{attribute 'OPC.UA.DA' := '1'}  				                
	{attribute 'OPC.UA.DA.Access' := '1'}  				                
	tb_Process_Complete													: BOOL;
	{attribute 'OPC.UA.DA' := '1'}  				                
	{attribute 'OPC.UA.DA.Access' := '1'}  				                
	tr_Remaining_Time													: REAL;
	{attribute 'OPC.UA.DA' := '1'}  				                
	{attribute 'OPC.UA.DA.Access' := '1'}  				                
	ti_Status															: INT;
	{attribute 'OPC.UA.DA' := '1'}  				                
	{attribute 'OPC.UA.DA.Access' := '1'}  				                
	ts_Status_Text														: STRING;		

	

	{attribute 'OPC.UA.DA' := '1'}  				                
	{attribute 'OPC.UA.DA.Access' := '1'}  				                
	interlock_inlet_door_clamps_or										: BOOL;

	{attribute 'OPC.UA.DA' := '1'}  				                
	{attribute 'OPC.UA.DA.Access' := '1'}  				                
	interlock_outlet_door_clamps_or										: BOOL;

	{attribute 'OPC.UA.DA' := '1'}  				                
	interlock_inlet_door_or												: BOOL;
	{attribute 'OPC.UA.DA' := '1'} 		      
	{attribute 'OPC.UA.DA.Access' := '1'}  				                
	interlock_inlet_door_or_status										: BOOL;
	{attribute 'OPC.UA.DA' := '1'}  				                
	{attribute 'OPC.UA.DA.Access' := '1'}  				                
	interlock_outlet_door_or											: BOOL;
	{attribute 'OPC.UA.DA' := '1'}  				                
	{attribute 'OPC.UA.DA.Access' := '1'}  				                
	interlock_outlet_door_or_status										: BOOL;
	
	{attribute 'OPC.UA.DA' := '1'}  				                
	interlock_inlet_door_clamp_or										: BOOL;
	{attribute 'OPC.UA.DA' := '1'}  				                
	{attribute 'OPC.UA.DA.Access' := '1'}  				                
	interlock_inlet_door_clamp_or_status								: BOOL;
	{attribute 'OPC.UA.DA' := '1'}  						                
	interlock_outlet_door_clamp_or										: BOOL;
	{attribute 'OPC.UA.DA' := '1'}  				                
	{attribute 'OPC.UA.DA.Access' := '1'}  				                
	interlock_outlet_door_clamp_or_status								: BOOL;
	
    /// <summary>PWR-01</summary>
	{attribute 'OPC.UA.DA' := '1'}  				                
	power_control														: BOOL;
    /// <summary>PWR-01</summary>
	{attribute 'OPC.UA.DA' := '1'}  				                
	{attribute 'OPC.UA.DA.Access' := '1'}  				                
	power_control_status												: BOOL;
    /// <summary>power_cmd</summary>
	PWR_01														AT %Q*	: BOOL;
	circuit_breaker_no_feedback									AT %I*	: BOOL;
	circuit_breaker_nc_feedback									AT %I*	: BOOL;
	

    /// <summary>RS_TT01</summary>
	{attribute 'OPC.UA.DA' := '1'}  				                
	{attribute 'OPC.UA.DA.Access' := '1'}  				                
	product_line_temp													: REAL;
    /// <summary>RS_TT01</summary>
	{attribute 'OPC.UA.DA' := '1'}  				                
	{attribute 'OPC.UA.DA.Access' := '1'}
	product_line_temp_error												: BOOL;
    /// <summary>RS_TT01</summary>
	{attribute 'OPC.UA.DA' := '1'}  				                
	_ProductLineTempErrorOff											: BOOL		:= TRUE;
    /// <summary>rs product line temp</summary>
	TT_01														AT %I*	: INT;
    /// <summary>rs product line temp</summary>
	TT_01_error													AT %I*	: BOOL;
	
    /// <summary>RS_PT02</summary>
	{attribute 'OPC.UA.DA' := '1'}  				                
	{attribute 'OPC.UA.DA.Access' := '1'}  				                
	product_line_pres													: REAL;
    /// <summary>RS_PT02</summary>
	{attribute 'OPC.UA.DA' := '1'}  				                
	{attribute 'OPC.UA.DA.Access' := '1'}  				                
	product_line_pres_error												: BOOL;
    /// <summary>RS_PT02</summary>
	{attribute 'OPC.UA.DA' := '1'}  				                
	_ProductLinePresErrorOff											: BOOL;
    /// <summary>rs product line temp</summary>
	PT_02														AT %I*	: INT;
    /// <summary>rs product line temp</summary>
	PT_02_error													AT %I*	: BOOL;
	
    /// <summary>RS_FT02</summary>
	{attribute 'OPC.UA.DA' := '1'}  				                
	{attribute 'OPC.UA.DA.Access' := '1'}  				                
	reactor_condensate_flow_error										: BOOL;
    /// <summary>RS_FT02</summary>
	{attribute 'OPC.UA.DA' := '1'}  				                
	_ReactorCondensateFlowErrorOff										: BOOL;
    /// <summary>rs reactor condensate flow</summary>
	FT_02														AT %I*	: INT;
    /// <summary>rs reactor condensate flow</summary>
	FT_02_error													AT %I*	: BOOL;

    /// <summary>RS_XV04</summary>
	{attribute 'OPC.UA.DA' := '1'}  				                
	dead_air_valve														: BOOL;
    /// <summary>RS_XV04</summary>
	{attribute 'OPC.UA.DA' := '1'}  				                
	{attribute 'OPC.UA.DA.Access' := '1'}  				                
	dead_air_valve_open_cmd_status										: BOOL;
    /// <summary>RS_XV04</summary>
	{attribute 'OPC.UA.DA' := '1'}  				                
	{attribute 'OPC.UA.DA.Access' := '1'}  				                
	dead_air_valve_open											AT %I*	: BOOL;
    /// <summary>RS_XV04</summary>
	{attribute 'OPC.UA.DA' := '1'}  				                
	{attribute 'OPC.UA.DA.Access' := '1'}  				                
	dead_air_valve_closed										AT %I*	: BOOL;
    /// <summary>dead air valve</summary>
	XV_04														AT %Q*	: BOOL;
	
    /// <summary>RS_XV05</summary>
	{attribute 'OPC.UA.DA' := '1'}  				                
	product_iso_valve													: BOOL;
    /// <summary>RS_XV05</summary>
	{attribute 'OPC.UA.DA' := '1'}  				                
	{attribute 'OPC.UA.DA.Access' := '1'}  				                
	product_iso_valve_open_cmd_status									: BOOL;
    /// <summary>RS_XV05</summary>
	{attribute 'OPC.UA.DA' := '1'}  				                
	{attribute 'OPC.UA.DA.Access' := '1'}  				                
	product_iso_valve_open										AT %I*	: BOOL;
    /// <summary>RS_XV05</summary>
	{attribute 'OPC.UA.DA' := '1'}  				                
	{attribute 'OPC.UA.DA.Access' := '1'}  				               
	product_iso_valve_closed									AT %I*	: BOOL;
    /// <summary>rs product iso valve</summary>
	XV_05														AT %Q*	: BOOL;
	
     /// <summary>RS_XV06</summary>
	{attribute 'OPC.UA.DA' := '1'}  				                
	condensate_valve													: BOOL;
    /// <summary>RS_XV06</summary>
	{attribute 'OPC.UA.DA' := '1'}  				                
	{attribute 'OPC.UA.DA.Access' := '1'}  				                
	condensate_valve_open_cmd_status									: BOOL;
    /// <summary>RS_XV06</summary>
	{attribute 'OPC.UA.DA' := '1'}  				                
	{attribute 'OPC.UA.DA.Access' := '1'}  				                
	condensate_valve_open										AT %I*	: BOOL;
    /// <summary>RS_XV06</summary>
	{attribute 'OPC.UA.DA' := '1'}  				                
	{attribute 'OPC.UA.DA.Access' := '1'}  				                
	condensate_valve_closed										AT %I*	: BOOL;
    /// <summary>cooling valve</summary>
	XV_06														AT %Q*	: BOOL;
	
    /// <summary>RS_XV07</summary>
	{attribute 'OPC.UA.DA' := '1'}  				                
	steam_iso_valve														: BOOL;
    /// <summary>RS_XV07</summary>
	{attribute 'OPC.UA.DA' := '1'}  				                
	{attribute 'OPC.UA.DA.Access' := '1'}  				                
	steam_iso_valve_open_cmd_status										: BOOL;
    /// <summary>RS_XV07</summary>
	{attribute 'OPC.UA.DA' := '1'}  				                
	{attribute 'OPC.UA.DA.Access' := '1'}  				                
	steam_iso_valve_closed										AT %I*	: BOOL;
    /// <summary>RS_XV07</summary>
	{attribute 'OPC.UA.DA' := '1'}  				                
	{attribute 'OPC.UA.DA.Access' := '1'}  				                
	steam_iso_valve_open										AT %I*	: BOOL;
    /// <summary>steam isolation valve</summary>
	XV_07														AT %Q*	: BOOL;

    /// <summary>RS_XV08</summary>
	{attribute 'OPC.UA.DA' := '1'}  				                
	{attribute 'OPC.UA.DA.Access' := '1'}  				                
	steam_bypass_valve_open_cmd_status									: BOOL;
    /// <summary>RS_XV08</summary>
	{attribute 'OPC.UA.DA' := '1'}  				                
	{attribute 'OPC.UA.DA.Access' := '1'}  				                
	steam_bypass_valve_open										AT %I*	: BOOL;
    /// <summary>RS_XV08</summary>
	{attribute 'OPC.UA.DA' := '1'}  				                
	{attribute 'OPC.UA.DA.Access' := '1'}  				                
	steam_bypass_valve_closed									AT %I*	: BOOL;
    /// <summary>steam bypass valve</summary>
	XV_08														AT %Q*	: BOOL;

	{attribute 'OPC.UA.DA' := '1'}  				                
	{attribute 'OPC.UA.DA.Access' := '1'}  				                
	reactor_test_leakage_pressure										: REAL;

END_VAR
VAR PERSISTENT
	
	{attribute 'OPC.UA.DA' := '1'}
	SP_include_inlet_doors_in_process									: BOOL;					
	{attribute 'OPC.UA.DA' := '1'}
	SP_include_outlet_doors_in_process									: BOOL;					

    /// <summary>TT01</summary>
	{attribute 'OPC.UA.DA' := '1'}  				                
	product_line_temp_offset											: REAL;

    /// <summary>PT02</summary>
	{attribute 'OPC.UA.DA' := '1'}  				                
	product_line_pres_low												: REAL;
    /// <summary>PT02</summary>
	{attribute 'OPC.UA.DA' := '1'}  				                
	product_line_pres_high												: REAL;
    /// <summary>PT02</summary>
	{attribute 'OPC.UA.DA' := '1'}  				                
	product_line_pres_min												: REAL;
    /// <summary>PT02</summary>
	{attribute 'OPC.UA.DA' := '1'}  				                
	product_line_pres_offset											: REAL;
	
    /// <summary>RS FT02</summary>
	{attribute 'OPC.UA.DA' := '1'}  				                
	reactor_condensate_flow_low											: REAL;
    /// <summary>RS FT02</summary>
	{attribute 'OPC.UA.DA' := '1'}  				                
	reactor_condensate_flow_high										: REAL;
    /// <summary>RS FT02</summary>
	{attribute 'OPC.UA.DA' := '1'}  				                
	reactor_condensate_flow_min											: REAL;
    /// <summary>RS FT02</summary>
	{attribute 'OPC.UA.DA' := '1'}  				                
	reactor_condensate_flow_offset										: REAL;
	
END_VAR

// Theseus - FB_Reactor_Set
// Rev 1.0 - December 2, 2024

r1(unit := 1);

A_Reactor_Set_IO();

IF eState <> eIdle THEN 
	A_Clear_Variables();
END_IF

iLength																	:= LEN(cycle_mode);
rtrigStart(CLK:= iLength > 0);
IF rtrigStart.Q THEN
	IF cycle_mode = '0' THEN
		bClearingCycle													:= TRUE;											// This acts as if the cycle ran so the reactor set cycle counter will stay in sync with the other reactor sets		
	ELSE
		bProcessStarted													:= TRUE;
		IF Pause_Reactor_Set THEN
			bPaused														:= TRUE;
		ELSE
			iStartStep													:= 1;
			Process_Running												:= TRUE;
			bMultiProcess												:= iLength > 1;
			giEvacuationCounter											:= 0;
			FOR i := 1 TO iLENGTH DO
				iStateMode[i]											:= STRING_TO_INT(MID(cycle_mode, 1, i));
				IF (iStateMode[i] = 6) THEN
					gbFirstEvacuation									:= TRUE;
					giEvacuationCounter									:= giEvacuationCounter + 1;
				END_IF
			END_FOR
			iStatePointer												:= 1;
			Machine_State												:= iStateMode[1];
		END_IF
	END_IF
END_IF

rtrigIdle(				CLK:= eState <= eIdle);
rtrigPaused(			CLk:= bPaused);
rtrigDoorCycle(			CLK:= Machine_State = eDoorCycle);
rtrigSingleProcessAuto(	CLK:= Machine_State = eSingleProcessAuto);
rtrigRepressurization(	CLK:= Machine_State = eRepressurization);
rtrigAdsorption(		CLK:= Machine_State = eAdsorption);
rtrigEvacuation(		CLK:= Machine_State = eEvacuation);
rtrigPositivePressure(	CLK:= Machine_State = ePositivePressure);
rtrigDesorption(		CLK:= Machine_State = eDesorption);
rtrigBypass(			CLK:= Machine_State = eBypass);

IF rtrigPaused.Q THEN
	bPaused																:= FALSE;
	eState																:= ePause;
ELSIF rtrigDoorCycle.Q THEN
	bDoorCycleDone														:= FALSE;
	i2Step																:= iStartStep;
	eState																:= eDoorCycle;
ELSIF rtrigPositivePressure.Q THEN
	bPositivePressureDone												:= FALSE;
	i3Step																:= iStartStep;
	eState																:= ePositivePressure;
ELSIF rtrigRepressurization.Q THEN
	bRepressurizationDone												:= FALSE;
	i4Step																:= iStartStep;
	eState																:= eRepressurization;
ELSIF rtrigAdsorption.Q THEN
	bAdsorptionDone														:= FALSE;
	i5Step																:= iStartStep;
	eState																:= eAdsorption;
ELSIF rtrigEvacuation.Q THEN
	bEvacuationDone														:= FALSE;
	i6Step																:= iStartStep;
	eState																:= eEvacuation;
ELSIF rtrigDesorption.Q THEN
	bDesorptionDone														:= FALSE;
	i7Step																:= iStartStep;
	eState																:= eDesorption;
ELSIF rtrigBypass.Q THEN
	bBypassDone															:= FALSE;
	i8Step																:= iStartStep;
	eState																:= eBypass;
ELSIF rtrigSingleProcessAuto.Q THEN
	eState																:= eSingleProcessAuto;
ELSIF rtrigIdle.Q THEN
	bProcessStarted														:= FALSE;
	eState																:= eIdle;
END_IF

CASE eState OF
	
	eIdle:
		A_Idle();
		
	eDoorCycle:
		IF bDoorCycleDone THEN
			DoorCycle_Running											:= FALSE;
			IF bMultiProcess THEN
				eState													:= SEL(bStop, eChangeState, ePause);
			ELSE
				Status													:= SEL(bStop, eDoorCycle_Complete, Status);
				eState													:= ePause;
			END_IF
		ELSIF bStop THEN
			Status														:= eStopping_Process;
		ELSE
			Status														:= eDoorCycle_Running;
			DoorCycle_Running											:= TRUE;
		END_IF
		
	ePositivePressure:
		IF bPositivePressureDone THEN
			PositivePressure_Running									:= FALSE;
			IF bMultiProcess THEN
				eState													:= SEL(bStop, eChangeState, ePause);
			ELSE
				Status													:= SEL(bStop, ePositivePressure_Complete, Status);
				eState													:= ePause;
			END_IF
		ELSIF bStop THEN
			Status														:= eStopping_Process;
		ELSE
			Status														:= ePositivePressure_Running;
			PositivePressure_Running									:= TRUE;
		END_IF

	eRepressurization:
		IF bRepressurizationDone THEN
			Repressurization_Running									:= FALSE;
			IF bMultiProcess THEN
				eState													:= SEL(bStop, eChangeState, ePause);
			ELSE
				Status													:= SEL(bStop, eRepressurization_Complete, Status);
				eState													:= ePause;
			END_IF
		ELSIF bStop THEN
			Status														:= eStopping_Process;
		ELSE
			Status														:= eRepressurization_Running;
			Repressurization_Running									:= TRUE;
		END_IF

	eAdsorption:
		IF bAdsorptionDone THEN
			Adsorption_Running											:= FALSE;
			IF bMultiProcess THEN
				eState													:= SEL(bStop, eChangeState, ePause);
			ELSE
				Status													:= SEL(bStop, eAdsorption_Complete, Status);
				eState													:= ePause;
			END_IF
		ELSIF bStop THEN
			Status														:= eStopping_Process;
		ELSE
			Status														:= eAdsorption_Running;
			Adsorption_Running											:= TRUE;
		END_IF

	eEvacuation:
		IF bEvacuationDone THEN
			Evacuation_Running											:= FALSE;
			IF bMultiProcess THEN
				eState													:= SEL(bStop, eChangeState, ePause);
			ELSE
				Status													:= SEL(bStop, eEvacuation_Complete, Status);
				eState													:= ePause;
			END_IF
		ELSIF bStop THEN
			Status														:= eStopping_Process;
		ELSE
			Status														:= eEvacuation_Running;
			Evacuation_Running											:= TRUE;
		END_IF
		
	eDesorption:
		IF bDesorptionDone THEN
			Desorption_Running											:= FALSE;
			IF bMultiProcess THEN
				eState													:= SEL(bStop, eChangeState, ePause);
			ELSE
				Status													:= SEL(bStop, eDesorption_Complete, Status);
				eState													:= ePause;
			END_IF
		ELSIF bStop THEN
			Status														:= eStopping_Process;
		ELSE
			Status														:= eDesorption_Running;
			Desorption_Running											:= TRUE;
		END_IF
		
	eBypass:
		IF bBypassDone THEN
			Bypass_Running												:= FALSE;
			IF bMultiProcess THEN
				eState													:= SEL(bStop, eChangeState, ePause);
			ELSE
				Status													:= SEL(bStop, eBypass_Complete, Status);
				eState													:= ePause;
			END_IF
		ELSIF bStop THEN
			Status														:= eStopping_Process;
		ELSE
			Status														:= eBypass_Running;
			Bypass_Running												:= TRUE;
		END_IF
		
	eSingleProcessAuto:
		eState															:= eChangeState;
		
	eChangeState:
		iStatePointer													:= iStatePointer + 1;
		IF iStatePointer > iLength THEN
			Process_Complete											:= TRUE;
			Done														:= TRUE;
			eState														:= eIdle;
		ELSIF iStateMode[iStatePointer] = 0 THEN
			Status														:= eStopping_Process;
			bStop														:= TRUE;
			bMultiProcess												:= FALSE;
			eState														:= ePause;
		ELSE
			Machine_State												:= iStateMode[iStatePointer];
		END_IF
	
	ePause:
		Machine_State													:= ePause;
		IF tonPause.Q THEN
			Done														:= TRUE;
			eState														:= eIdle;
		END_IF
		
END_CASE

bRunning																:= eState >= eRepressurization AND eState <= ePause;

A2_DoorCycle_1();
A3_PositivePressure_1();
A4_Repressurization_1();
A5_Adsorption_1();
A6_Evacuation_1();
A7_Desorption_1();
A8_Bypass_1();

(*
A4_Repressurization();
A5_Adsorption();
A6_Evacuation();
A7_Desorption();
A8_Bypass();
*)


A_Drain_Reactor_Set();

tonTimer1(IN:= bTimer1, PT:= REAL_TO_TIME(rTime1));
tonTimer2(IN:= bTimer2, PT:= REAL_TO_TIME(rTime2));
tonTimer3(IN:= bTimer3, PT:= REAL_TO_TIME(rTime3));

Remaining_Time															:= 0;
IF Process_Running THEN
	IF bTimer1 THEN
		Remaining_Time													:= rTime1 - TIME_TO_REAL(tonTimer1.ET);
	ELSIF bTimer2 THEN
		Remaining_Time													:= rTime2 - TIME_TO_REAL(tonTimer2.ET);
	ELSIF bTimer3 THEN
		Remaining_Time													:= rTime3 - TIME_TO_REAL(tonTimer3.ET);
	END_IF
END_IF

tonPause(IN:= eState = ePause, PT:= _TIMEOUT_RESET);
tonProcess(IN:= bProcessStarted, PT:= T#10H);

ti_Current_Step := Current_Step;
tr_Remaining_Time := Remaining_Time;
tb_Process_Running := Process_Running;

ACTION A_Check_Process:
// Theseus - FB_Reactor_Set.A_ClearProcess
// Rev 1.0 - June 13, 2024

Current_Step															:= iStep;
bEndProcess																:= FALSE;
IF stop_reactor_set THEN																									// Reactor Set can be stopped both internally and externally
	stop_reactor_set													:= FALSE;											// Clear flag
	bEndProcess															:= TRUE;											// Set flag to end process
ELSE
	IF sUtilityError <> '' THEN
		sError															:= sUtilityError;
		Utility_Error													:= TRUE;
		iStep															:= 98;
	ELSIF sReactorError <> '' THEN
		sError															:= sReactorError;
  		bEndProcess														:= TRUE;
	END_IF
	IF sError <> '' THEN
		P_Alarms.M_Add_Alarm(rs_name, F_Concat3(cycle_stage, ' ', sError), sMessage);
		sError															:= '';
	END_IF
END_IF

IF bEndProcess THEN
	bTimer1								 								:= FALSE;
	bTimer2								 								:= FALSE;
	bStop																:= TRUE;
	iStep																:= SEL(bMultiProcess, 80, 90);
END_IF
END_ACTION

ACTION A_Clear_Variables:
// Theseus - FB_Reactor_Set.A_Clear_Variables
// Rev 1.0 - November 26, 2024

//close_all_valves													:= FALSE;
//co2_sensors_on														:= FALSE;
Utility_Error															:= FALSE;
Cancel_Reactor_Set														:= FALSE;
Cancel_All_Reactor_Sets													:= FALSE;
sUtilityError															:= '';
sReactorError															:= '';
sRetryError																:= '';
IF clear_reactor_set_pause THEN
	clear_reactor_set_pause												:= FALSE;
	Pause_Reactor_Set													:= FALSE;
END_IF
IF NOT P_U01.auto_mode_on THEN
	iMaxSorbentTempErrorCount											:= 0;
	iCycleCount															:= 0;	
END_IF
END_ACTION

ACTION A_Drain_Reactor_Set:
// Theseus - FB_Reactor_Set.A_Drain_Reactor_Set
// Rev 1.0 - October 4, 2024

IF (gbDrainageOn OR P_U01.reactor_drain_or_on) AND NOT P_U01.reactor_drain_or_off THEN
	IF NOT r1.reactor_pres_error AND r1.reactor_pres >= P_U01.SP_minimum_drainage_pressure THEN
//		tonDrain(IN:= NOT bDrainError AND condensate_valve, PT:= REAL_TO_TIME(P_U01.SP_maximum_duration_to_drain_reactor_set * _SECONDS));
		IF tonDrain.Q AND reactor_condensate_flow < P_U01.SP_minimum_condensate_flow THEN
			condensate_valve											:= FALSE;
			IF TRUE THEN ///@@@reactor_drain_vessel_high THEN
				P_U01.steam_flow_control_valve							:= _CLOSED;
				P_Alarms.M_Add_Alarm(rs_name, gsReactorDrainError, gsMessageTBD);
				bDrainError												:= TRUE;
			END_IF
		ELSIF reactor_drain_vessel_lsh THEN ///@@@reactor_drain_vessel_high THEN							mm 11/7 
			condensate_valve											:= TRUE;
		ELSIF NOT reactor_drain_vessel_lsh AND NOT reactor_drain_vessel_lsl THEN ///@@@reactor_drain_vessel_low AND NOT reactor_drain_vessel_high THEN
			condensate_valve											:= FALSE;
//			bDrainError													:= FALSE;
		END_IF
	ELSE
//		IF NOT P_U01.reactor_drain_or_off  THEN 
			condensate_valve												:= FALSE;
//		END_IF
	END_IF
END_IF

rtrigCondensateValveOff_DrainOff(CLK := NOT gbDrainageOn AND NOT P_U01.reactor_drain_or_on AND NOT P_U01.reactor_drain_or_off);
IF 	rtrigCondensateValveOff_DrainOff.Q THEN
	condensate_valve												:= FALSE;
END_IF


gbCondensateValve														:= condensate_valve;

fb_adsorp_reactor_wastewater
	( i_execute := reactor_drain_adsorption_on,
	  i_value := P_U01.water_scale_3,
	  i_time := 30,
	  i_threshold := 1);
	  
IF reactor_drain_adsorption_on THEN
	IF NOT fb_adsorp_reactor_wastewater.o_below_threshold THEN
		condensate_valve											:= TRUE;
	ELSIF fb_adsorp_reactor_wastewater.o_below_threshold OR fb_adsorp_reactor_wastewater.o_timeout THEN
		condensate_valve											:= FALSE;
		reactor_drain_adsorption_on := FALSE;
	END_IF
END_IF
END_ACTION

ACTION A_Idle:
// Theseus - FB_Reactor_Set.A_Idle
// Rev 1.0 - June 24, 2024

Machine_State															:= eIdle;
cycle_stage																:= 'idle.idle';
sError																	:= '';
i4Step																	:= 0;
i5Step																	:= 0;
i6Step																	:= 0;
i7Step																	:= 0;
Current_Step															:= 0;
Remaining_Time															:= 0;
Current_Step															:= 0;
Status																	:= 0;
bMultiProcess															:= FALSE;
bTimer1																	:= FALSE;
bTimer2																	:= FALSE;
bStop																	:= FALSE;
Process_Running															:= FALSE;
Process_Complete														:= FALSE;
IF bClearingCycle THEN
	Done																:= TRUE;
	bClearingCycle														:= FALSE;
ELSE
	Done																:= FALSE;
END_IF
END_ACTION

ACTION A_Reactor_Set_IO:
// Theseus - A_Reactor_Set_IO
// Rev 1.0 - November 26, 2024

r1.fan_vfd_setpoint														:= fan_setpoint;

repres_valves_clear														:= r1.repres_valve_clear;

rAverageReactorPres														:= r1.reactor_pres;

//rso_power_control_out													:= rsi_power_control_fdbk_no AND NOT rsi_power_control_fdbk_nc AND NOT rso_PWR_01 ;
//rso_PWR_01																:= rsi_power_control_in;

interlock_inlet_door_or_status											:= interlock_inlet_door_or;
interlock_outlet_door_or_status											:= interlock_outlet_door_or;
interlock_inlet_door_clamp_or_status									:= interlock_inlet_door_clamp_or;
interlock_outlet_door_clamp_or_status									:= interlock_outlet_door_clamp_or;

inlet_doors_open														:= r1.inlet_doors_open;
inlet_doors_closed														:= r1.inlet_doors_closed;
outlet_doors_open														:= r1.outlet_doors_open;
outlet_doors_closed			 											:= r1.outlet_doors_closed;
 
gbGasketsActivated														:= SEL(NOT inlet_doors_closed OR NOT outlet_doors_closed, gbGasketsActivated, FALSE);					// PS 08_20_24

inlet_clamps_extended													:= r1.inlet_door_clamps_extended;
inlet_clamps_retracted													:= r1.inlet_door_clamps_retracted;
outlet_clamps_extended													:= r1.outlet_door_clamps_extended;
outlet_clamps_retracted													:= r1.outlet_door_clamps_retracted;

IF close_valves THEN
	dead_air_valve														:= FALSE;
	product_iso_valve													:= FALSE;
	condensate_valve													:= FALSE;
	steam_iso_valve														:= FALSE;
	steam_bypass_valve													:= FALSE;
	close_valves														:= FALSE;
END_IF

// Interlock 12
P_U01.door_open_with_steam_flow_interlock								:= NOT P_U01.steam_flow_control_valve_closed AND NOT steam_iso_valve_closed;
bCondition21															:= NOT P_U01.interlock_door_open_with_steam_flow_or AND P_U01.door_open_with_steam_flow_interlock;

// Interlock 14
P_U01.door_open_with_reactor_vacuum_interlock							:= rAverageReactorPres < 0.95;
bCondition22															:= NOT P_U01.interlock_door_open_with_reactor_vacuum_or AND P_U01.door_open_with_reactor_vacuum_interlock;

IF open_doors THEN
	r1.open_inlet_door													:= (inlet_clamps_retracted OR interlock_inlet_door_clamp_or)  AND NOT bCondition21 AND NOT bCondition22; // AND SP_include_inlet_doors_in_process;
	r1.open_outlet_door													:= (outlet_clamps_retracted OR interlock_outlet_door_clamp_or)  AND NOT bCondition21 AND NOT bCondition22; // AND SP_include_outlet_doors_in_process;
	open_doors															:= FALSE;
END_IF
IF close_doors THEN
	r1.close_inlet_door													:= (inlet_clamps_retracted OR interlock_inlet_door_clamp_or) ; //AND SP_include_inlet_doors_in_process;
	r1.close_outlet_door												:= (outlet_clamps_retracted OR interlock_outlet_door_clamp_or); // AND SP_include_outlet_doors_in_process;
	close_doors															:= FALSE;
END_IF

IF extend_clamps THEN
	r1.extend_inlet_door_clamps											:= (inlet_doors_closed OR interlock_inlet_door_or) AND SP_include_inlet_doors_in_process;
	r1.extend_outlet_door_clamps										:= (outlet_doors_closed OR interlock_outlet_door_or) AND SP_include_outlet_doors_in_process;
	extend_clamps														:= FALSE;
END_IF
IF retract_clamps THEN
	r1.retract_inlet_door_clamps										:= SP_include_inlet_doors_in_process;
	r1.retract_outlet_door_clamps										:= SP_include_outlet_doors_in_process;
	retract_clamps														:= FALSE;
END_IF

// CO2 adsorption sensor function
P_U01.co2_adsorption_interlock											:= r1.fan_vfd_setpoint > 10 AND r1.sorbent_high_temp < P_M01.SP_maximum_safe_co2_adsorption_sensor_temperature;
IF NOT P_U01.interlock_co2_adsorption_or THEN
	r1.inlet_co2_sol													:= P_U01.co2_adsorption_interlock;
	r1.outlet_co2_sol													:= P_U01.co2_adsorption_interlock;
	r1.outlet_co2_pump													:= TRUE;
	r1.inlet_co2_pump													:= TRUE;
ELSE
	r1.outlet_co2_pump													:= FALSE;
	r1.inlet_co2_pump													:= FALSE;
END_IF


r1.repres_valve															:= repres_valves AND gbRepresValves;

// Interlock 3
P_U01.hot_reactor_condenser_interlock									:= r1.temp_average > P_M01.SP_maximum_sorbent_temperature_to_use_dead_air_line;
IF NOT P_U01.interlock_hot_reactor_condenser_or and P_U01.hot_reactor_condenser_interlock THEN
	dead_air_valve														:= FALSE;
END_IF

XV_04																	:= dead_air_valve;
dead_air_valve_open_cmd_status											:= XV_04;
dead_air_valve_clear													:= F_ValveClear(dead_air_valve, dead_air_valve_open, dead_air_valve_closed);

XV_05																	:= product_iso_valve;
product_iso_valve_open_cmd_status										:= XV_05;
product_iso_valve_clear													:= F_ValveClear(product_iso_valve, product_iso_valve_open, product_iso_valve_closed);

XV_06																	:= condensate_valve;
condensate_valve_open_cmd_status										:= XV_06;
condensate_valve_clear													:= F_ValveClear(condensate_valve, condensate_valve_open, condensate_valve_closed);

// Interlock 4
P_U01.no_steam_unevacuated_reactor_interlock							:= r1.temp_high < P_M01.SP_maximum_safe_ambient_temperature AND NOT P_U01.steam_flow_control_valve_closed AND r1.reactor_pres < P_M01.SP_maximum_reactor_pressure_to_introduce_steam;
bCondition1																:= P_U01.interlock_no_steam_unevacuated_reactor_or OR P_U01.no_steam_unevacuated_reactor_interlock;

// Interlock 10
P_U01.reactor_over_safe_pressure_limit_interlock						:= r1.reactor_pres <= P_M01.SP_maximum_safe_reactor_steam_pressure;
bCondition2																:= P_U01.interlock_reactor_over_safe_pressure_limit_or OR P_U01.reactor_over_safe_pressure_limit_interlock;
r1.over_pressure_test_control											:= SEL(NOT bCondition2, r1.over_pressure_test_control, FALSE);

// Interlock 11
P_U01.reactor_over_safe_temperature_limit_interlock						:= r1.temp_high <= P_M01.SP_maximum_safe_sorbent_temperature;
bCondition3																:= P_U01.interlock_reactor_over_safe_temperature_limit_or OR P_U01.reactor_over_safe_temperature_limit_interlock;

IF NOT bCondition1 OR NOT bCondition2 OR NOT bCondition3 THEN
	steam_iso_valve														:= FALSE;
END_IF

XV_07																	:= steam_iso_valve;
steam_iso_valve_open_cmd_status											:= XV_07;
steam_iso_valve_clear													:= F_ValveClear(steam_iso_valve, steam_iso_valve_open, steam_iso_valve_closed);

XV_08																	:= steam_bypass_valve;
steam_bypass_valve_open_cmd_status										:= XV_08;
steam_bypass_valve_clear												:= F_ValveClear(steam_bypass_valve, steam_bypass_valve_open, steam_bypass_valve_closed);

rs_valves_clear															:= dead_air_valve_clear AND product_iso_valve_clear AND steam_iso_valve_clear AND steam_bypass_valve_clear AND condensate_valve_clear;

product_line_temp														:= F_Temperature(TT_01, product_line_temp_offset);
product_line_temp_error													:= TT_01_error AND NOT _ProductLineTempErrorOff;

product_line_pres														:= F_AnalogIn(PT_02, product_line_pres_low, product_line_pres_high, product_line_pres_min, product_line_pres_offset);
product_line_pres_error													:= PT_02_error AND NOT _ProductLinePresErrorOff;

reactor_condensate_flow													:= F_AnalogIn(FT_02, reactor_condensate_flow_low, reactor_condensate_flow_high, reactor_condensate_flow_min, reactor_condensate_flow_offset);
reactor_condensate_flow_error											:= FT_02_error AND NOT _ReactorCondensateFlowErrorOff;


gbCondenserKODrainageOn													:= product_line_pres >= P_U01.SP_minimum_drainage_pressure;

adsorption_high_temp_count												:= r1.adsorption_high_temp_count;
desorption_high_temp_count												:= r1.desorption_high_temp_count;
vacuum_cooling_high_temp_count											:= r1.vacuum_cooling_high_temp_count;
sorbent_high_temp														:= r1.sorbent_high_temp;
sorbent_average_temp													:= r1.sorbent_average_temp;

stop_reactor_set														:= stop_rs_automode;
stop_rs_automode														:= FALSE;
clear_reactor_set_pause													:= clear_rs_pause;
clear_rs_pause															:= FALSE;

//reactor_over_max_pressure												:= NOT r1.reactor_pres_error AND r1.reactor_pres > P_M01.SP_maximum_safe_reactor_steam_pressure;

rAveragePressure														:= 0;
iCount																	:= 0;
iVacuumStatus															:= 0;
iError																	:= 4;
IF NOT r1.reactor_pres_error THEN
	rAveragePressure													:= rAveragePressure + r1.reactor_pres;
	iVacuumStatus														:= F_LowMidHigh(r1.reactor_pres, P_M01.SP_target_desorption_starting_pressure, P_M01.SP_maximum_desorption_starting_pressure, iVacuumStatus);
	iCount																:= iCount + 1;
	iError																:= iError - 1;
END_IF
END_ACTION

ACTION A_Reset:
// Theseus - FB_Reactor_Set.A_Reset
// Rev 1.0 - November 25, 2024

r1.over_pressure_test_control											:= FALSE;
repres_valves															:= FALSE;
//co2_sensors_on														:= FALSE;
dead_air_valve															:= FALSE;
product_iso_valve														:= FALSE;
condensate_valve														:= FALSE;
steam_iso_valve															:= FALSE;
steam_bypass_valve														:= FALSE;
fan_setpoint															:= 0;
END_ACTION

ACTION A2_DoorCycle_1:
// Theseus - FB_Reactor_Set.A2_DoorCycle_1
// Rev 1.0 - June 26, 2024

CASE i2Step OF	

	0:	;
		
	1:
		cycle_stage														:= 'doorcycle.initialize';
		sMessage														:= gsSystemCannotRun;
		rTime1															:= 5 * _SECONDS;
		i2Step															:= i2Step + 1;
		
	2:
		bTimer1															:= TRUE;
		IF tonTimer1.Q THEN
			bTimer1														:= FALSE;
			i2Step														:= 99;
		END_IF
		
	99:
		bDoorCycleDone													:= TRUE;											// 9
		Current_Step													:= 0;
		i2Step															:= 0;
	
	
END_CASE

IF i2Step > 0 AND i2Step < 80 THEN
	iStep																:= i2Step;
	Current_Step														:= iStep;
	A_Check_Process();
	i2Step																:= iStep;
END_IF
END_ACTION

ACTION A2_DoorCycle_OLD:
// Theseus - FB_Reactor_Set.A2_DoorCycle
// Rev 1.0 - October 9, 2024

CASE i2Step OF	

	0:	;
		
	1:
		cycle_stage														:= 'doorcycle.initialize';
		sMessage														:= gsSystemCannotRun;
		IF NOT SP_include_inlet_doors_in_process AND NOT SP_include_outlet_doors_in_process THEN
			sReactorError												:= gsDoorsNotSelectedError;
		ELSIF r1.reactor_pres_error THEN
			sReactorError												:= gsReactorPresSensorError;
		ELSE
			A_Reset();																										// 1
			rTime1														:= 5 * _SECONDS;
			i2Step														:= i2Step + 1;
		END_IF
		
	2:
		bTimer1															:= TRUE;
		IF r1.reactor_pres > 0.98 AND r1.reactor_pres < 1.02 THEN															// 2
			bTimer1														:= FALSE;
			i2Step														:= i2Step + 1;
		ELSIF tonTimer1.Q THEN
			sReactorError												:= gsReactorNotAtAmbientPressure;
		END_IF
		
	3:
		bTimer1															:= TRUE;
		bPass1															:= bInletClampsRetracted;
		bPass2															:= bOutletClampsRetracted;
		IF bPass1 AND bPass2 THEN																							// 3
			bTimer1														:= FALSE;
			repres_valves												:= TRUE;											// 4
			rTime1														:= _VALVE_TIME;
			i2Step														:= i2Step + 1;
		ELSIF tonTimer1.Q THEN
			sReactorError												:= gsClampsNotRetractedError;
		END_IF
	
	4:
		bTimer1															:= TRUE;
		IF repres_valves_clear THEN
			cycle_stage													:= 'doorcycle.open';
			bTimer1														:= FALSE;
			open_doors													:= TRUE;											// 5
			rTime1														:= _DOOR_ACTUATION_TIMEOUT;
			i2Step														:= i2Step + 1;
		ELSIF tonTimer1.Q THEN
			sReactorError												:= gsRepressurizationValveError;
		END_IF
		
	5:
		bTimer1															:= TRUE;
		IF inlet_doors_open AND outlet_doors_open THEN
			bTimer1														:= FALSE;
			rTime1														:= 5 * _SECONDS;
			i2Step														:= i2Step + 1;
		ELSIF tonTimer1.Q THEN
			sReactorError												:= gsInletDoorNotOpenError;
			sReactorError												:= SEL(inlet_doors_open, gsOutletDoorNotOpenError, sReactorError);
		END_IF
		
	6:
		bTimer1															:= TRUE;
		IF tonTimer1.Q THEN																									// 6
			cycle_stage													:= 'doorcycle.close';
			bTimer1														:= FALSE;
			close_doors													:= TRUE;											// 7
			rTime1														:= _DOOR_ACTUATION_TIMEOUT;
			i2Step														:= i2Step + 1;
		END_IF
		
	7:
		bTimer1															:= TRUE;
		IF inlet_doors_closed AND outlet_doors_closed THEN
			bTimer1														:= FALSE;
			rTime1														:= 5 * _SECONDS;
			i2Step														:= i2Step + 1;
		ELSIF tonTimer1.Q THEN
			sReactorError												:= gsInletDoorNotClosedError;
			sReactorError												:= SEL(bPass2, gsOutletDoorNotClosedError, sReactorError);
		END_IF

	8:		
		bTimer1															:= TRUE;
		IF tonTimer1.Q THEN																									// 8
			bTimer1														:= FALSE;
			i2Step														:= 99;
		END_IF
	
	80:																														// Manual process closing
		cycle_stage														:= 'doorcycle.stopping';
		rTime1															:= _STOPPING_TIME;
		A_Reset();
		i2Step															:= 98;
		
	90:																														// Automatic process stopping
		cycle_stage														:= 'doorcycle.stopping';
		rTime1															:= _STOPPING_TIME;
		A_Reset();
		i2Step															:= 98;
		
	98:
		bTimer1															:= TRUE;
		IF tonTimer1.Q THEN
			bTimer1														:= FALSE;
			i2Step														:= 99;
		END_IF
		
	99:
		bDoorCycleDone													:= TRUE;											// 9
		Current_Step													:= 0;
		i2Step															:= 0;
	
	
END_CASE

IF i2Step > 0 AND i2Step < 80 THEN
	iStep																:= i2Step;
	Current_Step														:= iStep;
	A_Check_Process();
	i2Step																:= iStep;
END_IF
END_ACTION

ACTION A3_PositivePressure_1:
// Theseus - FB_Reactor_Set.A3_PositivePressure_1
// Rev 1.0 - June 26, 2024

CASE i3Step OF	

	0:	;
		
	1:
		cycle_stage														:= 'positivepressure.initialize';
		sMessage														:= gsSystemCannotRun;
		rTime1															:= _VALVE_TIME;
		i3Step															:= i3Step + 1;

	2:
		bTimer1															:= TRUE;
		IF tonTimer1.Q THEN
			bTimer1														:= FALSE;
			i3Step														:= 99;
		END_IF
	
	99:
		bPositivePressureDone											:= TRUE;
		Current_Step													:= 0;
		i3Step															:= 0;
	
	
END_CASE

IF i3Step > 0 AND i3Step < 80 THEN
	iStep																:= i3Step;
	Current_Step														:= iStep;
	A_Check_Process();
	i3Step																:= iStep;
END_IF
END_ACTION

ACTION A3_PositivePressure_OLD:
// Theseus - FB_Reactor_Set.A3_PositivePressure
// Rev 1.0 - October 3, 2024

CASE i3Step OF	

	0:	;
		
	1:
		cycle_stage														:= 'positivepressure.initialize';
		sMessage														:= gsSystemCannotRun;
		IF r1.reactor_pres_error THEN
			sReactorError												:= gsReactorPresSensorError;
		ELSE
			A_Reset();																										// 1
			i3Step														:= i3Step + 1;
		END_IF

	2:
		IF gbGasketsActivated THEN																							// 2
			rTime1														:= _VALVE_TIME;
			i3Step														:= i3Step + 1;
		ELSE
			sReactorError												:= gsGasketNotActivatedError;
		END_IF
		
	3:
		bTimer1															:= TRUE;
		IF repres_valves_clear AND rs_valves_clear THEN																	// 3
			bTimer1														:= FALSE;
			i3Step														:= i3Step + 1;
		ELSIF tonTimer1.Q THEN
			sReactorError												:= gsRepressurizationValveError;
			sReactorError												:= SEL(steam_iso_valve_clear, gsSteamIsoValveError, sReactorError);
			sReactorError												:= SEL(steam_bypass_valve_clear, gsSteamBypassValveError, sReactorError);
			sReactorError												:= SEL(product_iso_valve_clear, gsProductIsoValveError, sReactorError);
			sReactorError												:= SEL(dead_air_valve_clear, gsDeadAirValveError, sReactorError);
			sReactorError												:= SEL(condensate_valve_clear, gsCondensateValveError, sReactorError);
		END_IF
	
	4:
		IF bInletClampsExtended AND bOutletClampsExtended THEN																// 4
			cycle_stage													:= 'positivepressure.pressurizing';
			//m01_rs1_r1.XV_09											:= TRUE;											// smrg debug
			r1.over_pressure_test_control								:= TRUE;
			//overpressure_test_control								:= TRUE;											// 5
			rTime1														:= 5 * _MINUTES;
			i3Step														:= i3Step + 1;
		ELSE
			sReactorError												:= gsClampsNotExtendedError;
		END_IF
		
	5:
		bTimer1															:= TRUE;
		IF r1.reactor_pres >= P_M01.SP_pos_pres_ideal_pressure THEN
			bTimer1														:= FALSE;
			cycle_stage													:= 'positivepressure.settling';
			r1.over_pressure_test_control								:= FALSE;											// 6
			rTime1														:= P_M01.SP_pos_pres_settle_time * _MINUTES;		// 7
			i3Step														:= i3Step + 1;
		ELSIF tonTimer1.Q THEN
			sReactorError												:= gsPositivePressureError;
		END_IF
	
	6:
		bTimer1															:= TRUE;
		IF tonTimer1.Q THEN
			rR1SavedPressure											:= r1.reactor_pres;									// 8
			cycle_stage													:= 'positivepressure.leak_test';
			rTime1														:= P_M01.SP_pos_pres_leak_test_duration * _MINUTES;	// 9
			i3Step														:= i3Step + 1;
		END_IF
		
	7:
		bTimer1															:= TRUE;
		IF tonTimer1.Q THEN
			bTimer1														:= FALSE;
			rR1Leakage													:= (r1.reactor_pres - rR1SavedPressure) / P_M01.SP_pos_pres_leak_test_duration;	// 10
			IF rR1Leakage > P_M01.SP_unacceptable_pos_pres_change THEN
				sReactorError											:= gsUnacceptableReactorLeakRate;
			ELSE
				i3Step													:= 99;												// 11
			END_IF
		END_IF
		
	80:																														// Manual process closing
		cycle_stage														:= 'positivePressure.stopping';
		rTime1															:= _STOPPING_TIME;
		A_Reset();
		i3Step															:= 98;
		
	90:																														// Automatic process stopping
		cycle_stage														:= 'positivePressure.stopping';
		rTime1															:= _STOPPING_TIME;
		A_Reset();
		i3Step															:= 98;
		
	98:
		bTimer1															:= TRUE;
		IF tonTimer1.Q THEN
			bTimer1														:= FALSE;
			i3Step														:= 99;
		END_IF
		
	99:
		bPositivePressureDone											:= TRUE;
		Current_Step													:= 0;
		i3Step															:= 0;
	
	
END_CASE

IF i3Step > 0 AND i3Step < 80 THEN
	iStep																:= i3Step;
	Current_Step														:= iStep;
	A_Check_Process();
	i3Step																:= iStep;
END_IF
END_ACTION

ACTION A4_Repressurization:


CASE i4Step OF
	
	0:	;
	
	1: 
		cycle_stage														:= 'repressurization.initialize';
		sMessage														:= gsSystemCannotRun;
		
		IF P_U01.utility_error <> '' THEN
			sUtilityError												:= P_U01.utility_error;
		ELSIF r1.reactor_pres_error THEN
			sReactorError												:= gsReactorPresSensorError;
		ELSE			
//			A_Reset();
			P_U01.boiler_package 										:= FALSE;
			P_U01.steam_flow_control_valve_mode							:= eManual;
			P_U01.steam_flow_control_valve								:= _CLOSED;										
			dead_air_valve												:= FALSE;								// M01.XV04 <- FALSE
			product_iso_valve											:= FALSE;								// M01.XV05 <- FALSE
			steam_bypass_valve											:= FALSE;								// M01.XV08 <- FALSE
			rTime1														:= _VALVE_TIME;			
			i4Step														:= i4Step + 1;												
		END_IF		
		
	2: 
		cycle_stage														:= 'repressurization.starting';	
		bTimer1															:= TRUE;
		bPass1															:= P_U01.steam_flow_control_valve_closed;
		bPass2															:= dead_air_valve_closed;
		bPass3															:= product_iso_valve_clear;
		bPass4															:= steam_bypass_valve_clear;
		IF bPass1 AND bPass2 AND bPass3 AND bPass4  THEN
			bTimer1														:= FALSE; 
			i4Step														:= i4Step + 1;
		ELSIF tonTimer1.Q THEN
			bTimer1														:= FALSE; 
			sUtilityError												:= SEL(bPass1, gsSteamFlowConrolValveError, '');
			sReactorError												:= SEL(bPass2,gsDeadAirValveError,'');
			sReactorError												:= SEL(bPass3, gsProductIsoValveError, sReactorError);
			sReactorError												:= SEL(bPass1,'Steam Bypass Valve Error RS XV08', sReactorError);
		END_IF

	3: 
		bPass1 															:= sorbent_high_temp <= P_M01.SP_maximum_target_sorbent_temperature_to_repressurize;
		bPass2															:= r1.reactor_pres < 0.7;
		IF bPass1 AND bPass2 THEN
			rTime1														:= _CLAMP_ACTUATION_TIMEOUT;
			i4Step														:= i4Step + 1;
			
		ELSE
			sReactorError												:= SEL(bPass1,gsSorbentTemperatureError,'');
			sReactorError												:= SEL(bPass2,gsReactorPressureAboveDesiredLevelError,sReactorError);
		END_IF
		
	4: 
		
		bTimer1															:= TRUE;
		retract_clamps													:= TRUE;
		IF inlet_clamps_retracted AND outlet_clamps_retracted THEN 
			bTimer1														:= FALSE;
			repres_valves												:= TRUE;
			rTime1														:= _VALVE_TIME;
			rTime2														:= 5 * _SECONDS; 
			i4Step														:= i4Step + 1;	
		ELSIF tonTimer1.Q THEN
			bTimer1														:= FALSE; 
			sReactorError												:= gsDoorClampsExtendedError;
		END_IF
		
	5: 
		
		bTimer1															:= TRUE;
		
		IF r1.repres_valve_clear THEN 
			bTimer1														:= FALSE;
			bTimer2														:= TRUE;
			IF tonTimer2.Q THEN 
				bTimer2													:= FALSE;
				steam_iso_valve											:= TRUE;
				rTime1													:= _VALVE_TIME;
				i4Step													:= i4Step + 1;			
			END_IF
		ELSIF tonTimer1.Q THEN
			bTimer1														:= FALSE;
			bTimer2														:= FALSE;
			sReactorError												:= gsRepressurizationValveError;
		END_IF
		
	6: 
		
		bTimer1															:= TRUE;
		
		IF steam_iso_valve_clear THEN
			cycle_stage													:= 'repressurization.repressurize';
			bTimer1														:= FALSE;
			rTime1 														:= 2 * _MINUTES;
			i4Step														:= i4Step + 1;
		ELSIF tonTimer1.Q THEN
			bTimer1														:= FALSE;
			sReactorError												:= gsSteamIsoValveError;
		END_IF
		
	7: 
		
		bTimer1															:= TRUE;
		
		IF r1.reactor_pres > 0.98 AND r1.reactor_pres < 1.02 THEN															
			bTimer1														:= FALSE;
			rTime1														:= 10 * _SECONDS;
			i4Step														:= i4Step + 1;
		ELSIF tonTimer1.Q THEN
			bTimer1														:= FALSE;
			sReactorError												:= gsRepressurizationError;
		END_IF
		
		
	8: 
		
		bTimer1															:= TRUE;
		IF tonTimer1.Q THEN																									
			bTimer1														:= FALSE;
			repres_valves												:= FALSE;
			steam_iso_valve												:= FALSE;
			rTime1														:= _VALVE_TIME;
			i4Step														:= i4Step + 1;		
		END_IF
		
	9:
		
		bTimer1															:= TRUE;
	
		IF  r1.repres_valve_clear AND steam_iso_valve_clear THEN
			bTimer1														:= FALSE;
			rTime1														:= _STOPPING_TIME;
			i4Step														:= 98;
		ELSIF tonTimer1.Q THEN	
			bTimer1														:= FALSE;								
			sReactorError												:= SEL(r1.repres_valve_clear,gsRepressurizationValveError,'');
			sReactorError												:= SEL(steam_iso_valve_clear,gsSteamIsoValveError,sReactorError);

		END_IF
		
	
	80:																														// Manual process completing
		cycle_stage														:= 'repressurization.stopping';
		rTime1															:= _STOPPING_TIME;
		A_Reset();
		i4Step															:= 98;
		
	90:																														// Automatic process completing 
		cycle_stage														:= 'repressurization.stopping';
		rTime1															:= _STOPPING_TIME;
		A_Reset();
		i4Step															:= 98;
		
	98:
		bTimer1															:= TRUE;
		cycle_stage														:= 'repressurization.stopping';
		IF tonTimer1.Q THEN
			bTimer1														:= FALSE;
			i4Step														:= 99;
		END_IF
		
	99:
		bRepressurizationDone											:= TRUE;											// 5
		Current_Step													:= 0;
		i4Step															:= 0;
	
END_CASE

IF i4Step > 0 AND i4Step < 80 THEN
	iStep																:= i4Step;
	Current_Step														:= iStep;
	A_Check_Process();
	i4Step																:= iStep;
END_IF
END_ACTION

ACTION A4_Repressurization_1:
// Theseus - FB_Reactor_Set.A4_Repressurization_1
// Rev 1.0 - June 26, 2024

CASE i4Step OF
	
	0:	;
		
	1:
		cycle_stage														:= 'repressurization.initialize';
		rTime1															:= _VALVE_TIME;
		i4Step															:= i4Step + 1;
			
	2:
		cycle_stage														:= 'repressurization.running';
		bTimer1															:= TRUE;
		IF tonTimer1.Q THEN
			bTimer1														:= FALSE;
			i4Step														:= 98;
		END_IF
		
	80:																														// Manual process completing
		cycle_stage														:= 'repressurization.stopping.singlecycle';
		rTime1															:= _STOPPING_TIME;
		A_Reset();
		i4Step															:= 98;
		
	90:																														// Automatic process completing 
		cycle_stage														:= 'repressurization.stopping.multicycle';
		rTime1															:= _STOPPING_TIME;
		A_Reset();
		i4Step															:= 98;
		
	98:
		bTimer1															:= TRUE;
		//cycle_stage														:= 'repressurization.stopping';
		IF tonTimer1.Q THEN
			bTimer1														:= FALSE;
			i4Step														:= 99;
		END_IF
		

	99:
		bRepressurizationDone											:= TRUE;											// 5
		Current_Step													:= 0;
		i4Step															:= 0;
	
END_CASE

IF i4Step > 0 AND i4Step < 80 THEN
	iStep																:= i4Step;
	Current_Step														:= iStep;
	A_Check_Process();
	i4Step																:= iStep;
END_IF
END_ACTION

ACTION A4_Repressurization_OLD:
// Theseus - FB_Reactor_Set.A4_Repressurization
// Rev 1.0 - October 8, 2024

CASE i4Step OF
	
	0:	;
		
	1:
		cycle_stage														:= 'repressurization.initialize';
		sMessage														:= gsSystemCannotRun;
		IF P_U01.utility_error <> '' THEN
			sUtilityError												:= P_U01.utility_error;
		ELSIF r1.reactor_pres_error THEN
			sReactorError												:= gsReactorPresSensorError;
		ELSE
			A_Reset();																										// 1
			repres_valves												:= TRUE;											// 2		///@@@ Check clamps extended?
			steam_iso_valve												:= TRUE;
			rTime1														:= _VALVE_TIME;
			i4Step														:= i4Step + 1;
		END_IF
			
	2:
		bTimer1															:= TRUE;
		IF r1.repres_valve_clear AND steam_iso_valve_clear THEN
			bTimer1														:= FALSE;
			cycle_stage													:= 'repressurization.repressurize';
			rTime1														:= 5 * _MINUTES;
			i4Step														:= i4Step + 1;
		ELSIF tonTimer1.Q THEN
			sReactorError												:= SEL(r1.repres_valve_clear, gsRepressurizationValveError, gsSteamIsoValveError);
		END_IF

	3:
		bTimer1															:= TRUE;
		IF r1.reactor_pres > 0.98 AND r1.reactor_pres < 1.02 THEN															// 3
			bTimer1														:= FALSE;
			rTime1														:= 10 * _SECONDS;
			i4Step														:= i4Step + 1;
		ELSIF tonTimer1.Q THEN
			sReactorError												:= gsRepressurizationError;
		END_IF
		
	4:
		bTimer1															:= TRUE;
		IF tonTimer1.Q THEN																									// 4
			bTimer1														:= FALSE;
			i4Step														:= 99;
		END_IF
		
	
	80:																														// Manual process closing
		cycle_stage														:= 'repressurization.stopping';
		rTime1															:= _STOPPING_TIME;
		A_Reset();
		i4Step															:= 98;
		
	90:																														// Automatic process stopping
		cycle_stage														:= 'repressurization.stopping';
		rTime1															:= _STOPPING_TIME;
		A_Reset();
		i4Step															:= 98;
		
	98:
		bTimer1															:= TRUE;
		IF tonTimer1.Q THEN
			bTimer1														:= FALSE;
			i4Step														:= 99;
		END_IF
		
	99:
		bRepressurizationDone											:= TRUE;											// 5
		Current_Step													:= 0;
		i4Step															:= 0;
	
END_CASE

IF i4Step > 0 AND i4Step < 80 THEN
	iStep																:= i4Step;
	Current_Step														:= iStep;
	A_Check_Process();
	i4Step																:= iStep;
END_IF
END_ACTION

ACTION A5_Adsorption:
// Theseus - FB_Reactor_Set.A5_Adsorption
// Rev 1.0 - June 17, 2024

CASE i5Step OF	

	0:	;
		
	1:
		cycle_stage														:= 'adsorption.initialize';
		sMessage														:= gsSystemCannotRun;
		IF P_U01.utility_error <> '' THEN
			sUtilityError												:= P_U01.utility_error;
		ELSIF r1.reactor_pres_error THEN
			sReactorError												:= gsReactorPresSensorError;
		ELSE					
			retract_clamps												:= TRUE; 
			fan_setpoint												:= 0;
			steam_iso_valve												:= FALSE;      							// M01.XV07 <-TRUE
			P_U01.boiler_package 										:= FALSE;								// B01 : <- FALSE
			P_U01.steam_flow_control_valve_mode							:= eManual;
			P_U01.steam_flow_control_valve								:= _CLOSED;								// PCV02 <- CLOSE
			repres_valves												:= FALSE;								// R.XV02 <- TRUE
			dead_air_valve												:= FALSE;								// M01.XV04 <- FALSE
			steam_bypass_valve											:= FALSE;								// M01.XV08 <- FALSE
			product_iso_valve											:= FALSE;								// M01.XV05 <- FALSE
			P_U01.vacuum_pump_bypass_valve								:= TRUE;								// U01.XV04
			P_U01.product_line_ambient_valve							:= INT_TO_BOOL(eAmbient);				// U01.V11 <- ambient
			rTime1														:= 30 * _SECONDS;
			i5Step														:= i5Step + 1;												
		END_IF		
		
	2:
		
		bTimer1															:= TRUE;
		IF  inlet_clamps_retracted 					AND 
			outlet_clamps_retracted 				AND
			r1.fan_vfd_output = 0 					AND
			steam_iso_valve_clear					AND
			P_U01.steam_flow_control_valve_closed 	AND
			r1.repres_valve_clear					AND
			dead_air_valve_clear					AND
			steam_bypass_valve_clear				AND
			product_iso_valve_clear					AND
			P_U01.vacuum_pump_bypass_valve_clear 	AND
			P_U01.product_line_ambient_valve_clear 	AND 
			(r1.reactor_pres > 0.98 AND r1.reactor_pres < 1.02)  THEN
				
				bTimer1													:= FALSE; 
				rTime1													:= 5 * _SECONDS;
				i5Step													:= i5Step + 1; 
				
		ELSIF tonTimer1.Q THEN
			bTimer1														:= FALSE; 
			sReactorError												:= SEL(inlet_clamps_retracted,gsDoorClampsExtendedError,'');
			sReactorError												:= SEL(outlet_clamps_retracted,gsDoorClampsExtendedError,sReactorError);
			sReactorError												:= SEL(r1.fan_vfd_output <> 0,'fanVFDError',sReactorError);
			sReactorError												:= SEL(r1.repres_valve_clear,gsRepressurizationValveError,sReactorError);
			sReactorError												:= SEL(steam_iso_valve_clear,gsSteamIsoValveError,sReactorError);
			sReactorError												:= SEL(dead_air_valve_clear,gsDeadAirValveError,sReactorError);
			sReactorError												:= SEL(steam_bypass_valve_clear,gsSteamBypassValveError,sReactorError);
			sReactorError												:= SEL(product_iso_valve_clear,gsProductIsoValveError,sReactorError);
			sReactorError												:= SEL(r1.reactor_pres > 1.02, gsReactorPressureTooHighError ,sReactorError);
			sReactorError												:= SEL(r1.reactor_pres < 0.98, gsReactorPressureTooLowError ,sReactorError);
			
			sUtilityError												:= SEL(P_U01.vacuum_pump_bypass_valve_clear,'Vacuum Pump Bypass Valve Error ( U01.XV04)','');
			sUtilityError												:= SEL(P_U01.product_line_ambient_valve_clear,'Product Line Ambient Valve Error ( U01.XV11)',sUtilityError);
			sUtilityError												:= SEL(P_U01.steam_flow_control_valve_closed,gsSteamBypassValveError,sUtilityError);
		END_IF
		
	3: 
		bTimer1															:= TRUE;
		IF tonTimer1.Q THEN 
			bTimer1														:= FALSE;
			steam_iso_valve												:= TRUE;      							// M01.XV07 <-TRUE
			repres_valves												:= TRUE;								// R.XV02 <- TRUE
			rTime1														:= _VALVE_TIME;
			i5Step														:= i5Step + 1; 
		END_IF
		
	4: 
		bTimer1															:= TRUE;
		IF steam_iso_valve_clear AND r1.repres_valve_clear THEN
			bTimer1														:= FALSE;
			open_doors													:= TRUE;
			rTime1														:= _DOOR_ACTUATION_TIMEOUT;
			i5Step														:= i5Step + 1; 
		ELSIF tonTimer1.Q THEN
			bTimer1														:= FALSE;
			sReactorError												:= SEL(dead_air_valve_clear,gsDeadAirValveError,'');
			sReactorError												:= SEL(r1.repres_valve_clear,gsRepressurizationValveError,sReactorError);
		END_IF
		
		
	5: 
		
		bTimer1															:= TRUE;
			
		IF inlet_doors_open AND outlet_doors_open THEN	
			bTimer1														:= FALSE; 		
			fan_setpoint												:= P_M01.SP_reactor_set_1_vfd_percent;
			steam_iso_valve												:= FALSE; 
			repres_valves												:= FALSE;
			rTime1														:= _FAN_RS_DELAY_TIME;
			i5Step														:= i5Step + 1; 
		ELSIF tonTimer1.Q THEN
			bTimer1														:= FALSE; 
			sReactorError												:= gsDoorsNotOpenError;
		END_IF 
	
	6: 
		cycle_stage														:= 'adsorption.adsorption_started';
		bTimer1															:= TRUE;
		rTime2															:= P_M01.SP_adsorption_duration * _MINUTES;
		bTimer2															:= TRUE;
		bPass1															:= r1.fan_vfd_output >= fan_setpoint * 0.9 AND r1.fan_vfd_output <= fan_setpoint * 1.1;
		IF 	steam_iso_valve_clear AND
			r1.repres_valve_clear AND
			(r1.fan_vfd_output >= fan_setpoint * 0.9 AND r1.fan_vfd_output <= fan_setpoint * 1.1) THEN
			
				bTimer1													:= FALSE; 
				rTime1													:= 120 * _SECONDS;
				i5Step													:= i5Step + 1; 
				
		ELSIF tonTimer1.Q THEN
			bTimer1														:= FALSE; 
			sReactorError												:= SEL(bPass1,'Fan did not reach the set speed +/- 10%','');
			sReactorError												:= SEL(steam_iso_valve_clear,gsSteamControlValveError,sReactorError);
			sReactorError												:= SEL(r1.repres_valve_clear,gsRepressurizationValveError ,sReactorError);
		END_IF

	7: 
		
		bTimer1															:= TRUE;
		IF sorbent_average_temp < 40 THEN
			bTimer1														:= FALSE; 
			reactor_drain_adsorption_on									:= TRUE;
			rTime1														:= 120 * _SECONDS;
			i5Step														:= i5Step + 1; 
		ELSIF tonTimer1.Q THEN
			sReactorError												:= 'Evac Sorbent did not cool down enough at beginning of desorption';		
		END_IF
		
	8:   // new step
		
		IF NOT reactor_drain_adsorption_on THEN
			bTimer1														:= TRUE;
		END_IF
		IF tonTimer1.Q THEN
			bTimer1														:= FALSE;
			P_U01.condenser_knockout_drain_adsorption_on				:= TRUE;
			i5Step														:= i5Step + 1; 
		END_IF
		IF tonTimer2.Q THEN
			i5Step														:= i5Step + 1; 
		END_IF
		
	9: 
		
		IF tonTimer2.Q THEN
			bTimer2														:= FALSE; 
			fan_setpoint												:= 0;
			rTime1														:= 30 * _SECONDS;
			i5Step														:= i5Step + 1; 
		END_IF
		
	10: 
		
		
		bTimer1															:= TRUE;
		IF r1.fan_vfd_output = 0 AND tonTimer1.Q THEN
			bTimer1														:= FALSE; 
			close_doors													:= TRUE;
			rTime1														:= _DOOR_ACTUATION_TIMEOUT;
			i5Step														:= i5Step + 1; 
		ELSIF r1.fan_vfd_output <> 0 AND tonTimer1.Q THEN
			bTimer1														:= FALSE; 
			sReactorError												:= 'Adsorption Fan VFD did not turn off';	
		END_IF
		
	11:
		cycle_stage														:= 'adsorption.stopping ';
		
		bTimer1															:= TRUE;
		
		IF inlet_doors_closed AND outlet_doors_closed THEN
			bTimer1														:= FALSE; 
			P_U01.vacuum_pump_bypass_valve								:= FALSE;								// U01.XV04
			rTime1														:= _VALVE_TIME;
			i5Step														:= i5Step + 1; 
		
		ELSIF tonTimer1.Q THEN
			bTimer1														:= FALSE; 
			sReactorError												:= gsDoorsNotClosedError;
		END_IF
		
	12:
		
		bTimer1															:= TRUE;
				
		IF P_U01.vacuum_pump_bypass_valve_clear THEN
			bTimer1														:= FALSE; 
			rTime1														:= _STOPPING_TIME;
			i5Step														:= 98;
		ELSIF tonTimer1.Q THEN	
			bTimer1														:= FALSE; 	
			sReactorError												:= 'Vacuum Pump Bypass Error ( U01.XV04)';
		END_IF
		
	80:																														// Manual process completing
		cycle_stage														:= 'adsorption.stopping';
		rTime1															:= _STOPPING_TIME;
		A_Reset();
		i5Step															:= 98;
		
	90:																														// Automatic process completing 
		cycle_stage														:= 'adsorption.stopping';
		rTime1															:= _STOPPING_TIME;
		A_Reset();
		i5Step															:= 98;
		
	98:
		cycle_stage														:= 'adsorption.stopping';
		bTimer1															:= TRUE;
		IF tonTimer1.Q THEN
			bTimer1														:= FALSE;
			i5Step														:= 99;
		END_IF
		
	99:
		bAdsorptionDone													:= TRUE;											
		Current_Step													:= 0;
		i5Step															:= 0;	
	
END_CASE

IF i5Step > 0 AND i5Step < 80 THEN
	iStep																:= i5Step;
	Current_Step														:= iStep;
	A_Check_Process();
	i5Step																:= iStep;
END_IF
END_ACTION

ACTION A5_Adsorption_1:
// Theseus - FB_Reactor_Set.A5_Adsorption_1
// Rev 1.0 - June 26, 2024

CASE i5Step OF	

	0:	;
		
	1:
		cycle_stage														:= 'adsorption.initialize';
		rTime1															:= _VALVE_TIME;
		i5Step															:= i5Step + 1;
		
	2:
		cycle_stage														:= 'adsorption.initialize';
		bTimer1															:= TRUE;
		IF tonTimer1.Q THEN
			bTimer1														:= FALSE;
			i5Step														:= 98;
		END_IF
		
		
	80:																														// Manual process completing
		cycle_stage														:= 'adsorption.stopping';
		rTime1															:= _STOPPING_TIME;
		A_Reset();
		i5Step															:= 98;
		
	90:																														// Automatic process completing 
		cycle_stage														:= 'adsorption.stopping';
		rTime1															:= _STOPPING_TIME;
		A_Reset();
		i5Step															:= 98;
		
	98:
		cycle_stage														:= 'adsorption.stopping';
		bTimer1															:= TRUE;
		IF tonTimer1.Q THEN
			bTimer1														:= FALSE;
			i5Step														:= 99;
		END_IF
		
	
	99:
		cycle_stage														:= 'adsorption.completed';
		bAdsorptionDone													:= TRUE;											
		Current_Step													:= 0;
		i5Step															:= 0;
	
END_CASE

IF i5Step > 0 AND i5Step < 80 THEN
	iStep																:= i5Step;
	Current_Step														:= iStep;
	A_Check_Process();
	i5Step																:= iStep;
END_IF
END_ACTION

ACTION A5_Adsorption_OLD:
// Theseus - FB_Reactor_Set.A5_Adsorption
// Rev 1.0 - June 17, 2024

CASE i5Step OF	

	0:	;
		
	1:
		i5Step															:= 0;
	
END_CASE

IF i5Step > 0 AND i5Step < 80 THEN
	iStep																:= i5Step;
	Current_Step														:= iStep;
	A_Check_Process();
	i5Step																:= iStep;
END_IF
END_ACTION

ACTION A6_Evacuation:
// Theseus - FB_Reactor_Set.A6_Evacuation
// Rev 1.0 - December 3, 2024

CASE i6Step OF
	
	0:	;
	
	1:
		cycle_stage														:= 'evacuation.initialize';
		sMessage														:= gsSystemCannotRun;
		//gbGasketsActivated											:= FALSE;
		IF sorbent_high_temp < 60 THEN
			i6Step															:= i6Step + 1;										
		ELSE
			sReactorError												:= 'Sorbent too hot for dead air evacuation';
		END_IF
		
		
	2:
		//A_Reset();																											
		steam_bypass_valve												:= FALSE;								// M01.XV08 <- FALSE
		steam_iso_valve													:= FALSE;      							// M01.XV07 <-TRUE
		product_iso_valve												:= FALSE;								// M01.XV05 <- FALSE
		fan_setpoint													:= 0;
		P_U01.vacuum_pres_control_valve_mode							:= eManual;
		P_U01.vacuum_pres_control_valve									:= _CLOSED;
		P_U01.steam_flow_control_valve_mode								:= eManual;
		P_U01.steam_flow_control_valve									:= _CLOSED;
		P_U01.product_line_ambient_valve								:= FALSE;
		P_U01.vacuum_pump_bypass_valve									:= FALSE;								// U01.XV04
		P_U01.vacuum_pump_inlet_valve									:= FALSE;
//		P_U01.drainage_on												:= TRUE;
		rTime1															:= _VALVE_TIME;
		i6Step															:= i6Step + 1;
		
